   1:  PR[GP1:91,2] = PR[GP1:90,2] + 15.763;
   1:L PR[91] R[100]mm/sec CNT100;
   1:  PR[GP1:91,1] = PR[GP1:90,1] + -26.616;
   1:  PR[GP1:91,2] = PR[GP1:90,2] + 13.647;
   1:L PR[91] R[100]mm/sec CNT100;
   1:  PR[GP1:91,1] = PR[GP1:90,1] + -28.624;
   1:  PR[GP1:91,2] = PR[GP1:90,2] + 11.003;
   1:L PR[91] R[100]mm/sec CNT100;
   1:  PR[GP1:91,1] = PR[GP1:90,1] + -29.736;
   1:  PR[GP1:91,2] = PR[GP1:90,2] + 8.431;
   1:L PR[91] R[100]mm/sec CNT100;
   1:  PR[GP1:91,1] = PR[GP1:90,1] + -30.927;
   1:  PR[GP1:91,2] = PR[GP1:90,2] + 5.553;
   1:L PR[91] R[100]mm/sec CNT100;
   1:  PR[GP1:91,1] = PR[GP1:90,1] + -31.315;
   1:  PR[GP1:91,2] = PR[GP1:90,2] + 2.689;
   1:L PR[91] R[100]mm/sec CNT100;
   1:  PR[GP1:91,1] = PR[GP1:90,1] + -31.610;
   1:  PR[GP1:91,2] = PR[GP1:90,2] + -0.285;
   1:L PR[91] R[100]mm/sec CNT100;
   1:  PR[GP1:91,1] = PR[GP1:90,1] + -31.568;
   1:  PR[GP1:91,2] = PR[GP1:90,2] + -0.593;
   1:L PR[91] R[100]mm/sec CNT100;
   1:  PR[GP1:91,1] = PR[GP1:90,1] + -31.320;
   1:  PR[GP1:91,2] = PR[GP1:90,2] + -3.189;
   1:L PR[91] R[100]mm/sec CNT100;
   1:  PR[GP1:91,1] = PR[GP1:90,1] + -30.924;
   1:  PR[GP1:91,2] = PR[GP1:90,2] + -6.186;
   1:L PR[91] R[100]mm/sec CNT100;
   1:  PR[GP1:91,1] = PR[GP1:90,1] + -29.732;
   1:  PR[GP1:91,2] = PR[GP1:90,2] + -9.064;
   1:L PR[91] R[100]mm/sec CNT100;
   1:  PR[GP1:91,1] = PR[GP1:90,1] + -28.617;
   1:  PR[GP1:91,2] = PR[GP1:90,2] + -11.639;
   1:L PR[91] R[100]mm/sec CNT100;
   1:  PR[GP1:91,1] = PR[GP1:90,1] + -26.605;
   1:  PR[GP1:91,2] = PR[GP1:90,2] + -14.284;
   1:L PR[91] R[100]mm/sec CNT100;
   1:  PR[GP1:91,1] = PR[GP1:90,1] + -24.927;
   1:  PR[GP1:91,2] = PR[GP1:90,2] + -16.401;
   1:L PR[91] R[100]mm/sec CNT100;
   1:  PR[GP1:91,1] = PR[GP1:90,1] + -22.102;
   1:  PR[GP1:91,2] = PR[GP1:90,2] + -18.610;
   1:L PR[91] R[100]mm/sec CNT100;
   1:  PR[GP1:91,1] = PR[GP1:90,1] + -20.094;
   1:  PR[GP1:91,2] = PR[GP1:90,2] + -20.099;
   1:L PR[91] R[100]mm/sec CNT100;
   1:  PR[GP1:91,1] = PR[GP1:90,1] + -16.514;
   1:  PR[GP1:91,2] = PR[GP1:90,2] + -21.656;
   1:L PR[91] R[100]mm/sec CNT100;
   1:  PR[GP1:91,1] = PR[GP1:90,1] + -14.429;
   1:  PR[GP1:91,2] = PR[GP1:90,2] + -22.497;
   1:L PR[91] R[100]mm/sec CNT100;
   1:  PR[GP1:91,1] = PR[GP1:90,1] + -10.253;
   1:  PR[GP1:91,2] = PR[GP1:90,2] + -23.160;
   1:L PR[91] R[100]mm/sec CNT100;
   1:  PR[GP1:91,1] = PR[GP1:90,1] + -8.313;
   1:  PR[GP1:91,2] = PR[GP1:90,2] + -23.412;
   1:L PR[91] R[100]mm/sec CNT100;
   1:  PR[GP1:91,1] = PR[GP1:90,1] + -3.668;
   1:  PR[GP1:91,2] = PR[GP1:90,2] + -22.952;
   1:L PR[91] R[100]mm/sec CNT100;
   1:  PR[GP1:91,1] = PR[GP1:90,1] + -2.097;
   1:  PR[GP1:91,2] = PR[GP1:90,2] + -22.752;
   1:L PR[91] R[100]mm/sec CNT100;
   1:  PR[GP1:91,1] = PR[GP1:90,1] + -1.786;
   1:  PR[GP1:91,2] = PR[GP1:90,2] + -22.654;
   1:L PR[91] R[100]mm/sec CNT100;
   1:  PR[GP1:91,1] = PR[GP1:90,1] + -0.630;
   1:  PR[GP1:91,2] = PR[GP1:90,2] + -22.246;
   1:L PR[91] R[100]mm/sec CNT100;
   1:  PR[GP1:91,1] = PR[GP1:90,1] + 0.801;
   1:  PR[GP1:91,2] = PR[GP1:90,2] + -22.273;
   1:L PR[91] R[100]mm/sec CNT100;
   1:  PR[GP1:91,1] = PR[GP1:90,1] + 1.811;
   1:  PR[GP1:91,2] = PR[GP1:90,2] + -22.609;
   1:L PR[91] R[100]mm/sec CNT100;
   1:  PR[GP1:91,1] = PR[GP1:90,1] + 2.902;
   1:  PR[GP1:91,2] = PR[GP1:90,2] + -22.750;
   1:L PR[91] R[100]mm/sec CNT100;
   1:  PR[GP1:91,1] = PR[GP1:90,1] + 3.884;
   1:  PR[GP1:91,2] = PR[GP1:90,2] + -22.958;
   1:L PR[91] R[100]mm/sec CNT100;
   1:  PR[GP1:91,1] = PR[GP1:90,1] + 8.470;
   1:  PR[GP1:91,2] = PR[GP1:90,2] + -23.412;
   1:L PR[91] R[100]mm/sec CNT100;
   1:  PR[GP1:91,1] = PR[GP1:90,1] + 10.410;
   1:  PR[GP1:91,2] = PR[GP1:90,2] + -23.160;
   1:L PR[91] R[100]mm/sec CNT100;
   1:  PR[GP1:91,1] = PR[GP1:90,1] + 14.586;
   1:  PR[GP1:91,2] = PR[GP1:90,2] + -22.496;
   1:L PR[91] R[100]mm/sec CNT100;
   1:  PR[GP1:91,1] = PR[GP1:90,1] + 16.671;
   1:  PR[GP1:91,2] = PR[GP1:90,2] + -21.656;
   1:L PR[91] R[100]mm/sec CNT100;
   1:  PR[GP1:91,1] = PR[GP1:90,1] + 20.251;
   1:  PR[GP1:91,2] = PR[GP1:90,2] + -20.100;
   1:L PR[91] R[100]mm/sec CNT100;
   1:  PR[GP1:91,1] = PR[GP1:90,1] + 22.259;
   1:  PR[GP1:91,2] = PR[GP1:90,2] + -18.611;
   1:L PR[91] R[100]mm/sec CNT100;
   1:  PR[GP1:91,1] = PR[GP1:90,1] + 25.083;
   1:  PR[GP1:91,2] = PR[GP1:90,2] + -16.402;
   1:L PR[91] R[100]mm/sec CNT100;
   1:  PR[GP1:91,1] = PR[GP1:90,1] + 26.761;
   1:  PR[GP1:91,2] = PR[GP1:90,2] + -14.281;
   1:L PR[91] R[100]mm/sec CNT100;
   1:  PR[GP1:91,1] = PR[GP1:90,1] + 28.774;
   1:  PR[GP1:91,2] = PR[GP1:90,2] + -11.633;
   1:L PR[91] R[100]mm/sec CNT100;
   1:  PR[GP1:91,1] = PR[GP1:90,1] + 29.890;
   1:  PR[GP1:91,2] = PR[GP1:90,2] + -9.068;
   1:L PR[91] R[100]mm/sec CNT100;
   1:  PR[GP1:91,1] = PR[GP1:90,1] + 31.082;
   1:  PR[GP1:91,2] = PR[GP1:90,2] + -6.194;
   1:L PR[91] R[100]mm/sec CNT100;
   1:  PR[GP1:91,1] = PR[GP1:90,1] + 31.471;
   1:  PR[GP1:91,2] = PR[GP1:90,2] + -3.318;
   1:L PR[91] R[100]mm/sec CNT100;
   1:  PR[GP1:91,1] = PR[GP1:90,1] + 31.767;
   1:  PR[GP1:91,2] = PR[GP1:90,2] + -0.338;
   1:L PR[91] R[100]mm/sec CNT100;
   1:  PR[GP1:91,1] = PR[GP1:90,1] + 31.725;
   1:  PR[GP1:91,2] = PR[GP1:90,2] + -0.030;
   1:L PR[91] R[100]mm/sec CNT100;
   1:  PR[GP1:91,1] = PR[GP1:90,1] + 31.477;
   1:  PR[GP1:91,2] = PR[GP1:90,2] + 2.571;
   1:L PR[91] R[100]mm/sec CNT100;
   1:  PR[GP1:91,1] = PR[GP1:90,1] + 31.083;
   1:  PR[GP1:91,2] = PR[GP1:90,2] + 5.567;
   1:L PR[91] R[100]mm/sec CNT100;
   1:  PR[GP1:91,1] = PR[GP1:90,1] + 29.894;
   1:  PR[GP1:91,2] = PR[GP1:90,2] + 8.436;
   1:L PR[91] R[100]mm/sec CNT100;
   1:  PR[GP1:91,1] = PR[GP1:90,1] + 28.781;
   1:  PR[GP1:91,2] = PR[GP1:90,2] + 10.998;
   1:L PR[91] R[100]mm/sec CNT100;
   1:  PR[GP1:91,1] = PR[GP1:90,1] + 26.772;
   1:  PR[GP1:91,2] = PR[GP1:90,2] + 13.644;
   1:L PR[91] R[100]mm/sec CNT100;
   1:  PR[GP1:91,1] = PR[GP1:90,1] + 25.097;
   1:  PR[GP1:91,2] = PR[GP1:90,2] + 15.764;
   1:L PR[91] R[100]mm/sec CNT100;
   1:  PR[GP1:91,1] = PR[GP1:90,1] + 22.278;
   1:  PR[GP1:91,2] = PR[GP1:90,2] + 17.973;
   1:L PR[91] R[100]mm/sec CNT100;
   1:  PR[GP1:91,1] = PR[GP1:90,1] + 20.273;
   1:  PR[GP1:91,2] = PR[GP1:90,2] + 19.463;
   1:L PR[91] R[100]mm/sec CNT100;
   1:  PR[GP1:91,1] = PR[GP1:90,1] + 16.700;
   1:  PR[GP1:91,2] = PR[GP1:90,2] + 21.021;
   1:L PR[91] R[100]mm/sec CNT100;
   1:  PR[GP1:91,1] = PR[GP1:90,1] + 14.617;
   1:  PR[GP1:91,2] = PR[GP1:90,2] + 21.864;
   1:L PR[91] R[100]mm/sec CNT100;
   1:  PR[GP1:91,1] = PR[GP1:90,1] + 10.447;
   1:  PR[GP1:91,2] = PR[GP1:90,2] + 22.532;
   1:L PR[91] R[100]mm/sec CNT100;
   1:  PR[GP1:91,1] = PR[GP1:90,1] + 8.508;
   1:  PR[GP1:91,2] = PR[GP1:90,2] + 22.787;
   1:L PR[91] R[100]mm/sec CNT100;
   1:  PR[GP1:91,1] = PR[GP1:90,1] + 3.910;
   1:  PR[GP1:91,2] = PR[GP1:90,2] + 22.344;
   1:L PR[91] R[100]mm/sec CNT100;
   1:  PR[GP1:91,1] = PR[GP1:90,1] + 2.308;
   1:  PR[GP1:91,2] = PR[GP1:90,2] + 22.142;
   1:L PR[91] R[100]mm/sec CNT100;
   1:  PR[GP1:91,1] = PR[GP1:90,1] + 0.792;
   1:  PR[GP1:91,2] = PR[GP1:90,2] + 21.648;
   1:L PR[91] R[100]mm/sec CNT100;
   1:  PR[91] = PR[90];
   1:  PR[GP1:91,1] = PR[GP1:90,1] + -0.605;
   1:  PR[GP1:91,2] = PR[GP1:90,2] + 21.812;
   1:  PR[GP1:91,3] = PR[GP1:90,3] + 53.985;
   1:L PR[91] R[100]mm/sec CNT100;
   1:  PR[GP1:91,1] = PR[GP1:90,1] + -1.935;
   1:  PR[GP1:91,2] = PR[GP1:90,2] + 22.247;
   1:L PR[91] R[100]mm/sec CNT100;
   1:  PR[GP1:91,1] = PR[GP1:90,1] + -3.290;
   1:  PR[GP1:91,2] = PR[GP1:90,2] + 22.418;
   1:L PR[91] R[100]mm/sec CNT100;
   1:  PR[GP1:91,1] = PR[GP1:90,1] + -8.152;
   1:  PR[GP1:91,2] = PR[GP1:90,2] + 22.887;
   1:L PR[91] R[100]mm/sec CNT100;
   1:  PR[GP1:91,1] = PR[GP1:90,1] + -9.841;
   1:  PR[GP1:91,2] = PR[GP1:90,2] + 22.665;
   1:L PR[91] R[100]mm/sec CNT100;
   1:  PR[GP1:91,1] = PR[GP1:90,1] + -14.276;
   1:  PR[GP1:91,2] = PR[GP1:90,2] + 21.954;
   1:L PR[91] R[100]mm/sec CNT100;
   1:  PR[GP1:91,1] = PR[GP1:90,1] + -16.118;
   1:  PR[GP1:91,2] = PR[GP1:90,2] + 21.208;
   1:L PR[91] R[100]mm/sec CNT100;
   1:  PR[GP1:91,1] = PR[GP1:90,1] + -19.944;
   1:  PR[GP1:91,2] = PR[GP1:90,2] + 19.539;
   1:L PR[91] R[100]mm/sec CNT100;
   1:  PR[GP1:91,1] = PR[GP1:90,1] + -21.739;
   1:  PR[GP1:91,2] = PR[GP1:90,2] + 18.205;
   1:L PR[91] R[100]mm/sec CNT100;
   1:  PR[GP1:91,1] = PR[GP1:90,1] + -24.778;
   1:  PR[GP1:91,2] = PR[GP1:90,2] + 15.824;
   1:L PR[91] R[100]mm/sec CNT100;
   1:  PR[GP1:91,1] = PR[GP1:90,1] + -26.290;
   1:  PR[GP1:91,2] = PR[GP1:90,2] + 13.915;
   1:L PR[91] R[100]mm/sec CNT100;
   1:  PR[GP1:91,1] = PR[GP1:90,1] + -28.469;
   1:  PR[GP1:91,2] = PR[GP1:90,2] + 11.046;
   1:L PR[91] R[100]mm/sec CNT100;
   1:  PR[GP1:91,1] = PR[GP1:90,1] + -29.478;
   1:  PR[GP1:91,2] = PR[GP1:90,2] + 8.712;
   1:L PR[91] R[100]mm/sec CNT100;
   1:  PR[GP1:91,1] = PR[GP1:90,1] + -30.777;
   1:  PR[GP1:91,2] = PR[GP1:90,2] + 5.574;
   1:L PR[91] R[100]mm/sec CNT100;
   1:  PR[GP1:91,1] = PR[GP1:90,1] + -31.130;
   1:  PR[GP1:91,2] = PR[GP1:90,2] + 2.970;
   1:L PR[91] R[100]mm/sec CNT100;
   1:  PR[GP1:91,1] = PR[GP1:90,1] + -31.456;
   1:  PR[GP1:91,2] = PR[GP1:90,2] + -0.315;
   1:L PR[91] R[100]mm/sec CNT100;
   1:  PR[GP1:91,1] = PR[GP1:90,1] + -31.205;
   1:  PR[GP1:91,2] = PR[GP1:90,2] + -2.938;
   1:L PR[91] R[100]mm/sec CNT100;
   1:  PR[GP1:91,1] = PR[GP1:90,1] + -30.774;
   1:  PR[GP1:91,2] = PR[GP1:90,2] + -6.207;
   1:L PR[91] R[100]mm/sec CNT100;
   1:  PR[GP1:91,1] = PR[GP1:90,1] + -29.474;
   1:  PR[GP1:91,2] = PR[GP1:90,2] + -9.345;
   1:L PR[91] R[100]mm/sec CNT100;
   1:  PR[GP1:91,1] = PR[GP1:90,1] + -28.462;
   1:  PR[GP1:91,2] = PR[GP1:90,2] + -11.681;
   1:L PR[91] R[100]mm/sec CNT100;
   1:  PR[GP1:91,1] = PR[GP1:90,1] + -26.279;
   1:  PR[GP1:91,2] = PR[GP1:90,2] + -14.552;
   1:L PR[91] R[100]mm/sec CNT100;
   1:  PR[GP1:91,1] = PR[GP1:90,1] + -24.765;
   1:  PR[GP1:91,2] = PR[GP1:90,2] + -16.462;
   1:L PR[91] R[100]mm/sec CNT100;
   1:  PR[GP1:91,1] = PR[GP1:90,1] + -21.719;
   1:  PR[GP1:91,2] = PR[GP1:90,2] + -18.843;
   1:L PR[91] R[100]mm/sec CNT100;
   1:  PR[GP1:91,1] = PR[GP1:90,1] + -19.922;
   1:  PR[GP1:91,2] = PR[GP1:90,2] + -20.176;
   1:L PR[91] R[100]mm/sec CNT100;
   1:  PR[GP1:91,1] = PR[GP1:90,1] + -16.089;
   1:  PR[GP1:91,2] = PR[GP1:90,2] + -21.843;
   1:L PR[91] R[100]mm/sec CNT100;
   1:  PR[GP1:91,1] = PR[GP1:90,1] + -14.245;
   1:  PR[GP1:91,2] = PR[GP1:90,2] + -22.587;
   1:L PR[91] R[100]mm/sec CNT100;
   1:  PR[GP1:91,1] = PR[GP1:90,1] + -9.803;
   1:  PR[GP1:91,2] = PR[GP1:90,2] + -23.292;
   1:L PR[91] R[100]mm/sec CNT100;
   1:  PR[GP1:91,1] = PR[GP1:90,1] + -8.114;
   1:  PR[GP1:91,2] = PR[GP1:90,2] + -23.511;
   1:L PR[91] R[100]mm/sec CNT100;
   1:  PR[GP1:91,1] = PR[GP1:90,1] + -3.203;
   1:  PR[GP1:91,2] = PR[GP1:90,2] + -23.026;
   1:L PR[91] R[100]mm/sec CNT100;
   1:  PR[GP1:91,1] = PR[GP1:90,1] + -1.881;
   1:  PR[GP1:91,2] = PR[GP1:90,2] + -22.857;
   1:L PR[91] R[100]mm/sec CNT100;
   1:  PR[GP1:91,1] = PR[GP1:90,1] + -1.546;
   1:  PR[GP1:91,2] = PR[GP1:90,2] + -22.752;
   1:L PR[91] R[100]mm/sec CNT100;
   1:  PR[GP1:91,1] = PR[GP1:90,1] + -0.617;
   1:  PR[GP1:91,2] = PR[GP1:90,2] + -22.424;
   1:L PR[91] R[100]mm/sec CNT100;
   1:  PR[GP1:91,1] = PR[GP1:90,1] + 0.783;
   1:  PR[GP1:91,2] = PR[GP1:90,2] + -22.445;
   1:L PR[91] R[100]mm/sec CNT100;
   1:  PR[GP1:91,1] = PR[GP1:90,1] + 1.572;
   1:  PR[GP1:91,2] = PR[GP1:90,2] + -22.707;
   1:L PR[91] R[100]mm/sec CNT100;
   1:  PR[GP1:91,1] = PR[GP1:90,1] + 2.382;
   1:  PR[GP1:91,2] = PR[GP1:90,2] + -22.812;
   1:L PR[91] R[100]mm/sec CNT100;
   1:  PR[GP1:91,1] = PR[GP1:90,1] + 3.419;
   1:  PR[GP1:91,2] = PR[GP1:90,2] + -23.032;
   1:L PR[91] R[100]mm/sec CNT100;
   1:  PR[GP1:91,1] = PR[GP1:90,1] + 8.272;
   1:  PR[GP1:91,2] = PR[GP1:90,2] + -23.511;
   1:L PR[91] R[100]mm/sec CNT100;
   1:  PR[GP1:91,1] = PR[GP1:90,1] + 9.961;
   1:  PR[GP1:91,2] = PR[GP1:90,2] + -23.292;
   1:L PR[91] R[100]mm/sec CNT100;
   1:  PR[GP1:91,1] = PR[GP1:90,1] + 14.402;
   1:  PR[GP1:91,2] = PR[GP1:90,2] + -22.586;
   1:L PR[91] R[100]mm/sec CNT100;
   1:  PR[GP1:91,1] = PR[GP1:90,1] + 16.247;
   1:  PR[GP1:91,2] = PR[GP1:90,2] + -21.843;
   1:L PR[91] R[100]mm/sec CNT100;
   1:  PR[GP1:91,1] = PR[GP1:90,1] + 20.079;
   1:  PR[GP1:91,2] = PR[GP1:90,2] + -20.176;
   1:L PR[91] R[100]mm/sec CNT100;
   1:  PR[GP1:91,1] = PR[GP1:90,1] + 21.876;
   1:  PR[GP1:91,2] = PR[GP1:90,2] + -18.844;
   1:L PR[91] R[100]mm/sec CNT100;
   1:  PR[GP1:91,1] = PR[GP1:90,1] + 24.921;
   1:  PR[GP1:91,2] = PR[GP1:90,2] + -16.462;
   1:L PR[91] R[100]mm/sec CNT100;
   1:  PR[GP1:91,1] = PR[GP1:90,1] + 26.436;
   1:  PR[GP1:91,2] = PR[GP1:90,2] + -14.549;
   1:L PR[91] R[100]mm/sec CNT100;
   1:  PR[GP1:91,1] = PR[GP1:90,1] + 28.620;
   1:  PR[GP1:91,2] = PR[GP1:90,2] + -11.676;
   1:L PR[91] R[100]mm/sec CNT100;
   1:  PR[GP1:91,1] = PR[GP1:90,1] + 29.631;
   1:  PR[GP1:91,2] = PR[GP1:90,2] + -9.349;
   1:L PR[91] R[100]mm/sec CNT100;
   1:  PR[GP1:91,1] = PR[GP1:90,1] + 30.932;
   1:  PR[GP1:91,2] = PR[GP1:90,2] + -6.215;
   1:L PR[91] R[100]mm/sec CNT100;
   1:  PR[GP1:91,1] = PR[GP1:90,1] + 31.286;
   1:  PR[GP1:91,2] = PR[GP1:90,2] + -3.600;
   1:L PR[91] R[100]mm/sec CNT100;
   1:  PR[GP1:91,1] = PR[GP1:90,1] + 31.613;
   1:  PR[GP1:91,2] = PR[GP1:90,2] + -0.309;
   1:L PR[91] R[100]mm/sec CNT100;
   1:  PR[GP1:91,1] = PR[GP1:90,1] + 31.363;
   1:  PR[GP1:91,2] = PR[GP1:90,2] + 2.319;
   1:L PR[91] R[100]mm/sec CNT100;
   1:  PR[GP1:91,1] = PR[GP1:90,1] + 30.932;
   1:  PR[GP1:91,2] = PR[GP1:90,2] + 5.587;
   1:L PR[91] R[100]mm/sec CNT100;
   1:  PR[GP1:91,1] = PR[GP1:90,1] + 29.635;
   1:  PR[GP1:91,2] = PR[GP1:90,2] + 8.716;
   1:L PR[91] R[100]mm/sec CNT100;
   1:  PR[GP1:91,1] = PR[GP1:90,1] + 28.626;
   1:  PR[GP1:91,2] = PR[GP1:90,2] + 11.041;
   1:L PR[91] R[100]mm/sec CNT100;
   1:  PR[GP1:91,1] = PR[GP1:90,1] + 26.446;
   1:  PR[GP1:91,2] = PR[GP1:90,2] + 13.912;
   1:L PR[91] R[100]mm/sec CNT100;
   1:  PR[GP1:91,1] = PR[GP1:90,1] + 24.934;
   1:  PR[GP1:91,2] = PR[GP1:90,2] + 15.825;
   1:L PR[91] R[100]mm/sec CNT100;
   1:  PR[GP1:91,1] = PR[GP1:90,1] + 21.896;
   1:  PR[GP1:91,2] = PR[GP1:90,2] + 18.206;
   1:L PR[91] R[100]mm/sec CNT100;
   1:  PR[GP1:91,1] = PR[GP1:90,1] + 20.101;
   1:  PR[GP1:91,2] = PR[GP1:90,2] + 19.540;
   1:L PR[91] R[100]mm/sec CNT100;
   1:  PR[GP1:91,1] = PR[GP1:90,1] + 16.275;
   1:  PR[GP1:91,2] = PR[GP1:90,2] + 21.208;
   1:L PR[91] R[100]mm/sec CNT100;
   1:  PR[GP1:91,1] = PR[GP1:90,1] + 14.433;
   1:  PR[GP1:91,2] = PR[GP1:90,2] + 21.953;
   1:L PR[91] R[100]mm/sec CNT100;
   1:  PR[GP1:91,1] = PR[GP1:90,1] + 9.998;
   1:  PR[GP1:91,2] = PR[GP1:90,2] + 22.665;
   1:L PR[91] R[100]mm/sec CNT100;
   1:  PR[GP1:91,1] = PR[GP1:90,1] + 8.309;
   1:  PR[GP1:91,2] = PR[GP1:90,2] + 22.887;
   1:L PR[91] R[100]mm/sec CNT100;
   1:  PR[GP1:91,1] = PR[GP1:90,1] + 3.448;
   1:  PR[GP1:91,2] = PR[GP1:90,2] + 22.418;
   1:L PR[91] R[100]mm/sec CNT100;
   1:  PR[GP1:91,1] = PR[GP1:90,1] + 2.090;
   1:  PR[GP1:91,2] = PR[GP1:90,2] + 22.247;
   1:L PR[91] R[100]mm/sec CNT100;
   1:  PR[GP1:91,1] = PR[GP1:90,1] + 0.770;
   1:  PR[GP1:91,2] = PR[GP1:90,2] + 21.820;
   1:L PR[91] R[100]mm/sec CNT100;
   1:  PR[91] = PR[90];
   1:  PR[GP1:91,1] = PR[GP1:90,1] + -0.589;
   1:  PR[GP1:91,2] = PR[GP1:90,2] + 21.992;
   1:  PR[GP1:91,3] = PR[GP1:90,3] + 54.595;
   1:L PR[91] R[100]mm/sec CNT100;
   1:  PR[GP1:91,1] = PR[GP1:90,1] + -1.714;
   1:  PR[GP1:91,2] = PR[GP1:90,2] + 22.352;
   1:L PR[91] R[100]mm/sec CNT100;
   1:  PR[GP1:91,1] = PR[GP1:90,1] + -2.827;
   1:  PR[GP1:91,2] = PR[GP1:90,2] + 22.492;
   1:L PR[91] R[100]mm/sec CNT100;
   1:  PR[GP1:91,1] = PR[GP1:90,1] + -7.953;
   1:  PR[GP1:91,2] = PR[GP1:90,2] + 22.986;
   1:L PR[91] R[100]mm/sec CNT100;
   1:  PR[GP1:91,1] = PR[GP1:90,1] + -9.391;
   1:  PR[GP1:91,2] = PR[GP1:90,2] + 22.797;
   1:L PR[91] R[100]mm/sec CNT100;
   1:  PR[GP1:91,1] = PR[GP1:90,1] + -14.091;
   1:  PR[GP1:91,2] = PR[GP1:90,2] + 22.044;
   1:L PR[91] R[100]mm/sec CNT100;
   1:  PR[GP1:91,1] = PR[GP1:90,1] + -15.693;
   1:  PR[GP1:91,2] = PR[GP1:90,2] + 21.395;
   1:L PR[91] R[100]mm/sec CNT100;
   1:  PR[GP1:91,1] = PR[GP1:90,1] + -19.772;
   1:  PR[GP1:91,2] = PR[GP1:90,2] + 19.616;
   1:L PR[91] R[100]mm/sec CNT100;
   1:  PR[GP1:91,1] = PR[GP1:90,1] + -21.356;
   1:  PR[GP1:91,2] = PR[GP1:90,2] + 18.438;
   1:L PR[91] R[100]mm/sec CNT100;
   1:  PR[GP1:91,1] = PR[GP1:90,1] + -24.616;
   1:  PR[GP1:91,2] = PR[GP1:90,2] + 15.885;
   1:L PR[91] R[100]mm/sec CNT100;
   1:  PR[GP1:91,1] = PR[GP1:90,1] + -25.964;
   1:  PR[GP1:91,2] = PR[GP1:90,2] + 14.182;
   1:L PR[91] R[100]mm/sec CNT100;
   1:  PR[GP1:91,1] = PR[GP1:90,1] + -28.314;
   1:  PR[GP1:91,2] = PR[GP1:90,2] + 11.088;
   1:L PR[91] R[100]mm/sec CNT100;
   1:  PR[GP1:91,1] = PR[GP1:90,1] + -29.220;
   1:  PR[GP1:91,2] = PR[GP1:90,2] + 8.993;
   1:L PR[91] R[100]mm/sec CNT100;
   1:  PR[GP1:91,1] = PR[GP1:90,1] + -30.626;
   1:  PR[GP1:91,2] = PR[GP1:90,2] + 5.595;
   1:L PR[91] R[100]mm/sec CNT100;
   1:  PR[GP1:91,1] = PR[GP1:90,1] + -30.944;
   1:  PR[GP1:91,2] = PR[GP1:90,2] + 3.251;
   1:L PR[91] R[100]mm/sec CNT100;
   1:  PR[GP1:91,1] = PR[GP1:90,1] + -31.251;
   1:  PR[GP1:91,2] = PR[GP1:90,2] + 0.151;
   1:L PR[91] R[100]mm/sec CNT100;
   1:  PR[GP1:91,1] = PR[GP1:90,1] + -31.315;
   1:  PR[GP1:91,2] = PR[GP1:90,2] + -0.338;
   1:L PR[91] R[100]mm/sec CNT100;
   1:  PR[GP1:91,1] = PR[GP1:90,1] + -31.091;
   1:  PR[GP1:91,2] = PR[GP1:90,2] + -2.686;
   1:L PR[91] R[100]mm/sec CNT100;
   1:  PR[GP1:91,1] = PR[GP1:90,1] + -30.623;
   1:  PR[GP1:91,2] = PR[GP1:90,2] + -6.228;
   1:L PR[91] R[100]mm/sec CNT100;
   1:  PR[GP1:91,1] = PR[GP1:90,1] + -29.215;
   1:  PR[GP1:91,2] = PR[GP1:90,2] + -9.626;
   1:L PR[91] R[100]mm/sec CNT100;
   1:  PR[GP1:91,1] = PR[GP1:90,1] + -28.307;
   1:  PR[GP1:91,2] = PR[GP1:90,2] + -11.724;
   1:L PR[91] R[100]mm/sec CNT100;
   1:  PR[GP1:91,1] = PR[GP1:90,1] + -25.953;
   1:  PR[GP1:91,2] = PR[GP1:90,2] + -14.819;
   1:L PR[91] R[100]mm/sec CNT100;
   1:  PR[GP1:91,1] = PR[GP1:90,1] + -24.602;
   1:  PR[GP1:91,2] = PR[GP1:90,2] + -16.522;
   1:L PR[91] R[100]mm/sec CNT100;
   1:  PR[GP1:91,1] = PR[GP1:90,1] + -21.336;
   1:  PR[GP1:91,2] = PR[GP1:90,2] + -19.076;
   1:L PR[91] R[100]mm/sec CNT100;
   1:  PR[GP1:91,1] = PR[GP1:90,1] + -19.750;
   1:  PR[GP1:91,2] = PR[GP1:90,2] + -20.253;
   1:L PR[91] R[100]mm/sec CNT100;
   1:  PR[GP1:91,1] = PR[GP1:90,1] + -15.664;
   1:  PR[GP1:91,2] = PR[GP1:90,2] + -22.030;
   1:L PR[91] R[100]mm/sec CNT100;
   1:  PR[GP1:91,1] = PR[GP1:90,1] + -14.061;
   1:  PR[GP1:91,2] = PR[GP1:90,2] + -22.677;
   1:L PR[91] R[100]mm/sec CNT100;
   1:  PR[GP1:91,1] = PR[GP1:90,1] + -9.354;
   1:  PR[GP1:91,2] = PR[GP1:90,2] + -23.424;
   1:L PR[91] R[100]mm/sec CNT100;
   1:  PR[GP1:91,1] = PR[GP1:90,1] + -7.915;
   1:  PR[GP1:91,2] = PR[GP1:90,2] + -23.611;
   1:L PR[91] R[100]mm/sec CNT100;
   1:  PR[GP1:91,1] = PR[GP1:90,1] + -2.738;
   1:  PR[GP1:91,2] = PR[GP1:90,2] + -23.099;
   1:L PR[91] R[100]mm/sec CNT100;
   1:  PR[GP1:91,1] = PR[GP1:90,1] + -1.676;
   1:  PR[GP1:91,2] = PR[GP1:90,2] + -22.963;
   1:L PR[91] R[100]mm/sec CNT100;
   1:  PR[GP1:91,1] = PR[GP1:90,1] + -0.592;
   1:  PR[GP1:91,2] = PR[GP1:90,2] + -22.602;
   1:L PR[91] R[100]mm/sec CNT100;
   1:  PR[GP1:91,1] = PR[GP1:90,1] + 0.765;
   1:  PR[GP1:91,2] = PR[GP1:90,2] + -22.616;
   1:L PR[91] R[100]mm/sec CNT100;
   1:  PR[GP1:91,1] = PR[GP1:90,1] + 1.333;
   1:  PR[GP1:91,2] = PR[GP1:90,2] + -22.805;
   1:L PR[91] R[100]mm/sec CNT100;
   1:  PR[GP1:91,1] = PR[GP1:90,1] + 1.862;
   1:  PR[GP1:91,2] = PR[GP1:90,2] + -22.874;
   1:L PR[91] R[100]mm/sec CNT100;
   1:  PR[GP1:91,1] = PR[GP1:90,1] + 2.955;
   1:  PR[GP1:91,2] = PR[GP1:90,2] + -23.105;
   1:L PR[91] R[100]mm/sec CNT100;
   1:  PR[GP1:91,1] = PR[GP1:90,1] + 8.073;
   1:  PR[GP1:91,2] = PR[GP1:90,2] + -23.611;
   1:L PR[91] R[100]mm/sec CNT100;
   1:  PR[GP1:91,1] = PR[GP1:90,1] + 9.512;
   1:  PR[GP1:91,2] = PR[GP1:90,2] + -23.424;
   1:L PR[91] R[100]mm/sec CNT100;
   1:  PR[GP1:91,1] = PR[GP1:90,1] + 14.218;
   1:  PR[GP1:91,2] = PR[GP1:90,2] + -22.676;
   1:L PR[91] R[100]mm/sec CNT100;
   1:  PR[GP1:91,1] = PR[GP1:90,1] + 15.823;
   1:  PR[GP1:91,2] = PR[GP1:90,2] + -22.030;
   1:L PR[91] R[100]mm/sec CNT100;
   1:  PR[GP1:91,1] = PR[GP1:90,1] + 19.907;
   1:  PR[GP1:91,2] = PR[GP1:90,2] + -20.253;
   1:L PR[91] R[100]mm/sec CNT100;
   1:  PR[GP1:91,1] = PR[GP1:90,1] + 21.493;
   1:  PR[GP1:91,2] = PR[GP1:90,2] + -19.077;
   1:L PR[91] R[100]mm/sec CNT100;
   1:  PR[GP1:91,1] = PR[GP1:90,1] + 24.759;
   1:  PR[GP1:91,2] = PR[GP1:90,2] + -16.523;
   1:L PR[91] R[100]mm/sec CNT100;
   1:  PR[GP1:91,1] = PR[GP1:90,1] + 26.110;
   1:  PR[GP1:91,2] = PR[GP1:90,2] + -14.816;
   1:L PR[91] R[100]mm/sec CNT100;
   1:  PR[GP1:91,1] = PR[GP1:90,1] + 28.465;
   1:  PR[GP1:91,2] = PR[GP1:90,2] + -11.718;
   1:L PR[91] R[100]mm/sec CNT100;
   1:  PR[GP1:91,1] = PR[GP1:90,1] + 29.373;
   1:  PR[GP1:91,2] = PR[GP1:90,2] + -9.630;
   1:L PR[91] R[100]mm/sec CNT100;
   1:  PR[GP1:91,1] = PR[GP1:90,1] + 30.781;
   1:  PR[GP1:91,2] = PR[GP1:90,2] + -6.235;
   1:L PR[91] R[100]mm/sec CNT100;
   1:  PR[GP1:91,1] = PR[GP1:90,1] + 31.100;
   1:  PR[GP1:91,2] = PR[GP1:90,2] + -3.881;
   1:L PR[91] R[100]mm/sec CNT100;
   1:  PR[GP1:91,1] = PR[GP1:90,1] + 31.408;
   1:  PR[GP1:91,2] = PR[GP1:90,2] + -0.776;
   1:L PR[91] R[100]mm/sec CNT100;
   1:  PR[GP1:91,1] = PR[GP1:90,1] + 31.472;
   1:  PR[GP1:91,2] = PR[GP1:90,2] + -0.286;
   1:L PR[91] R[100]mm/sec CNT100;
   1:  PR[GP1:91,1] = PR[GP1:90,1] + 31.248;
   1:  PR[GP1:91,2] = PR[GP1:90,2] + 2.066;
   1:L PR[91] R[100]mm/sec CNT100;
   1:  PR[GP1:91,1] = PR[GP1:90,1] + 30.782;
   1:  PR[GP1:91,2] = PR[GP1:90,2] + 5.608;
   1:L PR[91] R[100]mm/sec CNT100;
   1:  PR[GP1:91,1] = PR[GP1:90,1] + 29.377;
   1:  PR[GP1:91,2] = PR[GP1:90,2] + 8.997;
   1:L PR[91] R[100]mm/sec CNT100;
   1:  PR[GP1:91,1] = PR[GP1:90,1] + 28.471;
   1:  PR[GP1:91,2] = PR[GP1:90,2] + 11.083;
   1:L PR[91] R[100]mm/sec CNT100;
   1:  PR[GP1:91,1] = PR[GP1:90,1] + 26.120;
   1:  PR[GP1:91,2] = PR[GP1:90,2] + 14.180;
   1:L PR[91] R[100]mm/sec CNT100;
   1:  PR[GP1:91,1] = PR[GP1:90,1] + 24.772;
   1:  PR[GP1:91,2] = PR[GP1:90,2] + 15.886;
   1:L PR[91] R[100]mm/sec CNT100;
   1:  PR[GP1:91,1] = PR[GP1:90,1] + 21.513;
   1:  PR[GP1:91,2] = PR[GP1:90,2] + 18.439;
   1:L PR[91] R[100]mm/sec CNT100;
   1:  PR[GP1:91,1] = PR[GP1:90,1] + 19.929;
   1:  PR[GP1:91,2] = PR[GP1:90,2] + 19.617;
   1:L PR[91] R[100]mm/sec CNT100;
   1:  PR[GP1:91,1] = PR[GP1:90,1] + 15.851;
   1:  PR[GP1:91,2] = PR[GP1:90,2] + 21.395;
   1:L PR[91] R[100]mm/sec CNT100;
   1:  PR[GP1:91,1] = PR[GP1:90,1] + 14.248;
   1:  PR[GP1:91,2] = PR[GP1:90,2] + 22.043;
   1:L PR[91] R[100]mm/sec CNT100;
   1:  PR[GP1:91,1] = PR[GP1:90,1] + 9.549;
   1:  PR[GP1:91,2] = PR[GP1:90,2] + 22.797;
   1:L PR[91] R[100]mm/sec CNT100;
   1:  PR[GP1:91,1] = PR[GP1:90,1] + 8.110;
   1:  PR[GP1:91,2] = PR[GP1:90,2] + 22.986;
   1:L PR[91] R[100]mm/sec CNT100;
   1:  PR[GP1:91,1] = PR[GP1:90,1] + 2.985;
   1:  PR[GP1:91,2] = PR[GP1:90,2] + 22.492;
   1:L PR[91] R[100]mm/sec CNT100;
   1:  PR[GP1:91,1] = PR[GP1:90,1] + 1.872;
   1:  PR[GP1:91,2] = PR[GP1:90,2] + 22.351;
   1:L PR[91] R[100]mm/sec CNT100;
   1:  PR[GP1:91,1] = PR[GP1:90,1] + 0.749;
   1:  PR[GP1:91,2] = PR[GP1:90,2] + 21.992;
   1:L PR[91] R[100]mm/sec CNT100;
   1:  PR[91] = PR[90];
   1:  PR[GP1:91,1] = PR[GP1:90,1] + -0.574;
   1:  PR[GP1:91,2] = PR[GP1:90,2] + 22.162;
   1:  PR[GP1:91,3] = PR[GP1:90,3] + 55.205;
   1:L PR[91] R[100]mm/sec CNT100;
   1:  PR[GP1:91,1] = PR[GP1:90,1] + -1.497;
   1:  PR[GP1:91,2] = PR[GP1:90,2] + 22.457;
   1:L PR[91] R[100]mm/sec CNT100;
   1:  PR[GP1:91,1] = PR[GP1:90,1] + -2.364;
   1:  PR[GP1:91,2] = PR[GP1:90,2] + 22.566;
   1:L PR[91] R[100]mm/sec CNT100;
   1:  PR[GP1:91,1] = PR[GP1:90,1] + -7.753;
   1:  PR[GP1:91,2] = PR[GP1:90,2] + 23.086;
   1:L PR[91] R[100]mm/sec CNT100;
   1:  PR[GP1:91,1] = PR[GP1:90,1] + -8.942;
   1:  PR[GP1:91,2] = PR[GP1:90,2] + 22.929;
   1:L PR[91] R[100]mm/sec CNT100;
   1:  PR[GP1:91,1] = PR[GP1:90,1] + -13.907;
   1:  PR[GP1:91,2] = PR[GP1:90,2] + 22.134;
   1:L PR[91] R[100]mm/sec CNT100;
   1:  PR[GP1:91,1] = PR[GP1:90,1] + -15.269;
   1:  PR[GP1:91,2] = PR[GP1:90,2] + 21.582;
   1:L PR[91] R[100]mm/sec CNT100;
   1:  PR[GP1:91,1] = PR[GP1:90,1] + -19.600;
   1:  PR[GP1:91,2] = PR[GP1:90,2] + 19.693;
   1:L PR[91] R[100]mm/sec CNT100;
   1:  PR[GP1:91,1] = PR[GP1:90,1] + -20.974;
   1:  PR[GP1:91,2] = PR[GP1:90,2] + 18.672;
   1:L PR[91] R[100]mm/sec CNT100;
   1:  PR[GP1:91,1] = PR[GP1:90,1] + -24.454;
   1:  PR[GP1:91,2] = PR[GP1:90,2] + 15.946;
   1:L PR[91] R[100]mm/sec CNT100;
   1:  PR[GP1:91,1] = PR[GP1:90,1] + -25.638;
   1:  PR[GP1:91,2] = PR[GP1:90,2] + 14.449;
   1:L PR[91] R[100]mm/sec CNT100;
   1:  PR[GP1:91,1] = PR[GP1:90,1] + -28.159;
   1:  PR[GP1:91,2] = PR[GP1:90,2] + 11.131;
   1:L PR[91] R[100]mm/sec CNT100;
   1:  PR[GP1:91,1] = PR[GP1:90,1] + -28.962;
   1:  PR[GP1:91,2] = PR[GP1:90,2] + 9.274;
   1:L PR[91] R[100]mm/sec CNT100;
   1:  PR[GP1:91,1] = PR[GP1:90,1] + -30.476;
   1:  PR[GP1:91,2] = PR[GP1:90,2] + 5.616;
   1:L PR[91] R[100]mm/sec CNT100;
   1:  PR[GP1:91,1] = PR[GP1:90,1] + -30.758;
   1:  PR[GP1:91,2] = PR[GP1:90,2] + 3.532;
   1:L PR[91] R[100]mm/sec CNT100;
   1:  PR[GP1:91,1] = PR[GP1:90,1] + -31.034;
   1:  PR[GP1:91,2] = PR[GP1:90,2] + 0.748;
   1:L PR[91] R[100]mm/sec CNT100;
   1:  PR[GP1:91,1] = PR[GP1:90,1] + -31.177;
   1:  PR[GP1:91,2] = PR[GP1:90,2] + -0.338;
   1:L PR[91] R[100]mm/sec CNT100;
   1:  PR[GP1:91,1] = PR[GP1:90,1] + -30.976;
   1:  PR[GP1:91,2] = PR[GP1:90,2] + -2.434;
   1:L PR[91] R[100]mm/sec CNT100;
   1:  PR[GP1:91,1] = PR[GP1:90,1] + -30.473;
   1:  PR[GP1:91,2] = PR[GP1:90,2] + -6.249;
   1:L PR[91] R[100]mm/sec CNT100;
   1:  PR[GP1:91,1] = PR[GP1:90,1] + -28.957;
   1:  PR[GP1:91,2] = PR[GP1:90,2] + -9.907;
   1:L PR[91] R[100]mm/sec CNT100;
   1:  PR[GP1:91,1] = PR[GP1:90,1] + -28.152;
   1:  PR[GP1:91,2] = PR[GP1:90,2] + -11.766;
   1:L PR[91] R[100]mm/sec CNT100;
   1:  PR[GP1:91,1] = PR[GP1:90,1] + -25.627;
   1:  PR[GP1:91,2] = PR[GP1:90,2] + -15.086;
   1:L PR[91] R[100]mm/sec CNT100;
   1:  PR[GP1:91,1] = PR[GP1:90,1] + -24.440;
   1:  PR[GP1:91,2] = PR[GP1:90,2] + -16.583;
   1:L PR[91] R[100]mm/sec CNT100;
   1:  PR[GP1:91,1] = PR[GP1:90,1] + -20.954;
   1:  PR[GP1:91,2] = PR[GP1:90,2] + -19.309;
   1:L PR[91] R[100]mm/sec CNT100;
   1:  PR[GP1:91,1] = PR[GP1:90,1] + -19.578;
   1:  PR[GP1:91,2] = PR[GP1:90,2] + -20.330;
   1:L PR[91] R[100]mm/sec CNT100;
   1:  PR[GP1:91,1] = PR[GP1:90,1] + -15.240;
   1:  PR[GP1:91,2] = PR[GP1:90,2] + -22.217;
   1:L PR[91] R[100]mm/sec CNT100;
   1:  PR[GP1:91,1] = PR[GP1:90,1] + -13.876;
   1:  PR[GP1:91,2] = PR[GP1:90,2] + -22.767;
   1:L PR[91] R[100]mm/sec CNT100;
   1:  PR[GP1:91,1] = PR[GP1:90,1] + -8.905;
   1:  PR[GP1:91,2] = PR[GP1:90,2] + -23.557;
   1:L PR[91] R[100]mm/sec CNT100;
   1:  PR[GP1:91,1] = PR[GP1:90,1] + -7.716;
   1:  PR[GP1:91,2] = PR[GP1:90,2] + -23.710;
   1:L PR[91] R[100]mm/sec CNT100;
   1:  PR[GP1:91,1] = PR[GP1:90,1] + -2.273;
   1:  PR[GP1:91,2] = PR[GP1:90,2] + -23.172;
   1:L PR[91] R[100]mm/sec CNT100;
   1:  PR[GP1:91,1] = PR[GP1:90,1] + -1.456;
   1:  PR[GP1:91,2] = PR[GP1:90,2] + -23.068;
   1:L PR[91] R[100]mm/sec CNT100;
   1:  PR[GP1:91,1] = PR[GP1:90,1] + -0.575;
   1:  PR[GP1:91,2] = PR[GP1:90,2] + -22.780;
   1:L PR[91] R[100]mm/sec CNT100;
   1:  PR[GP1:91,1] = PR[GP1:90,1] + 0.746;
   1:  PR[GP1:91,2] = PR[GP1:90,2] + -22.787;
   1:L PR[91] R[100]mm/sec CNT100;
   1:  PR[GP1:91,1] = PR[GP1:90,1] + 1.094;
   1:  PR[GP1:91,2] = PR[GP1:90,2] + -22.903;
   1:L PR[91] R[100]mm/sec CNT100;
   1:  PR[GP1:91,1] = PR[GP1:90,1] + 1.342;
   1:  PR[GP1:91,2] = PR[GP1:90,2] + -22.935;
   1:L PR[91] R[100]mm/sec CNT100;
   1:  PR[GP1:91,1] = PR[GP1:90,1] + 2.490;
   1:  PR[GP1:91,2] = PR[GP1:90,2] + -23.178;
   1:L PR[91] R[100]mm/sec CNT100;
   1:  PR[GP1:91,1] = PR[GP1:90,1] + 7.874;
   1:  PR[GP1:91,2] = PR[GP1:90,2] + -23.711;
   1:L PR[91] R[100]mm/sec CNT100;
   1:  PR[GP1:91,1] = PR[GP1:90,1] + 9.063;
   1:  PR[GP1:91,2] = PR[GP1:90,2] + -23.557;
   1:L PR[91] R[100]mm/sec CNT100;
   1:  PR[GP1:91,1] = PR[GP1:90,1] + 14.034;
   1:  PR[GP1:91,2] = PR[GP1:90,2] + -22.766;
   1:L PR[91] R[100]mm/sec CNT100;
   1:  PR[GP1:91,1] = PR[GP1:90,1] + 15.398;
   1:  PR[GP1:91,2] = PR[GP1:90,2] + -22.216;
   1:L PR[91] R[100]mm/sec CNT100;
   1:  PR[GP1:91,1] = PR[GP1:90,1] + 19.735;
   1:  PR[GP1:91,2] = PR[GP1:90,2] + -20.330;
   1:L PR[91] R[100]mm/sec CNT100;
   1:  PR[GP1:91,1] = PR[GP1:90,1] + 21.111;
   1:  PR[GP1:91,2] = PR[GP1:90,2] + -19.310;
   1:L PR[91] R[100]mm/sec CNT100;
   1:  PR[GP1:91,1] = PR[GP1:90,1] + 24.597;
   1:  PR[GP1:91,2] = PR[GP1:90,2] + -16.584;
   1:L PR[91] R[100]mm/sec CNT100;
   1:  PR[GP1:91,1] = PR[GP1:90,1] + 25.784;
   1:  PR[GP1:91,2] = PR[GP1:90,2] + -15.084;
   1:L PR[91] R[100]mm/sec CNT100;
   1:  PR[GP1:91,1] = PR[GP1:90,1] + 28.310;
   1:  PR[GP1:91,2] = PR[GP1:90,2] + -11.761;
   1:L PR[91] R[100]mm/sec CNT100;
   1:  PR[GP1:91,1] = PR[GP1:90,1] + 29.115;
   1:  PR[GP1:91,2] = PR[GP1:90,2] + -9.910;
   1:L PR[91] R[100]mm/sec CNT100;
   1:  PR[GP1:91,1] = PR[GP1:90,1] + 30.631;
   1:  PR[GP1:91,2] = PR[GP1:90,2] + -6.256;
   1:L PR[91] R[100]mm/sec CNT100;
   1:  PR[GP1:91,1] = PR[GP1:90,1] + 30.914;
   1:  PR[GP1:91,2] = PR[GP1:90,2] + -4.163;
   1:L PR[91] R[100]mm/sec CNT100;
   1:  PR[GP1:91,1] = PR[GP1:90,1] + 31.190;
   1:  PR[GP1:91,2] = PR[GP1:90,2] + -1.374;
   1:L PR[91] R[100]mm/sec CNT100;
   1:  PR[GP1:91,1] = PR[GP1:90,1] + 31.333;
   1:  PR[GP1:91,2] = PR[GP1:90,2] + -0.286;
   1:L PR[91] R[100]mm/sec CNT100;
   1:  PR[GP1:91,1] = PR[GP1:90,1] + 31.133;
   1:  PR[GP1:91,2] = PR[GP1:90,2] + 1.814;
   1:L PR[91] R[100]mm/sec CNT100;
   1:  PR[GP1:91,1] = PR[GP1:90,1] + 30.631;
   1:  PR[GP1:91,2] = PR[GP1:90,2] + 5.628;
   1:L PR[91] R[100]mm/sec CNT100;
   1:  PR[GP1:91,1] = PR[GP1:90,1] + 29.119;
   1:  PR[GP1:91,2] = PR[GP1:90,2] + 9.277;
   1:L PR[91] R[100]mm/sec CNT100;
   1:  PR[GP1:91,1] = PR[GP1:90,1] + 28.316;
   1:  PR[GP1:91,2] = PR[GP1:90,2] + 11.126;
   1:L PR[91] R[100]mm/sec CNT100;
   1:  PR[GP1:91,1] = PR[GP1:90,1] + 25.795;
   1:  PR[GP1:91,2] = PR[GP1:90,2] + 14.447;
   1:L PR[91] R[100]mm/sec CNT100;
   1:  PR[GP1:91,1] = PR[GP1:90,1] + 24.610;
   1:  PR[GP1:91,2] = PR[GP1:90,2] + 15.946;
   1:L PR[91] R[100]mm/sec CNT100;
   1:  PR[GP1:91,1] = PR[GP1:90,1] + 21.131;
   1:  PR[GP1:91,2] = PR[GP1:90,2] + 18.672;
   1:L PR[91] R[100]mm/sec CNT100;
   1:  PR[GP1:91,1] = PR[GP1:90,1] + 19.757;
   1:  PR[GP1:91,2] = PR[GP1:90,2] + 19.693;
   1:L PR[91] R[100]mm/sec CNT100;
   1:  PR[GP1:91,1] = PR[GP1:90,1] + 15.427;
   1:  PR[GP1:91,2] = PR[GP1:90,2] + 21.582;
   1:L PR[91] R[100]mm/sec CNT100;
   1:  PR[GP1:91,1] = PR[GP1:90,1] + 14.064;
   1:  PR[GP1:91,2] = PR[GP1:90,2] + 22.133;
   1:L PR[91] R[100]mm/sec CNT100;
   1:  PR[GP1:91,1] = PR[GP1:90,1] + 9.100;
   1:  PR[GP1:91,2] = PR[GP1:90,2] + 22.930;
   1:L PR[91] R[100]mm/sec CNT100;
   1:  PR[GP1:91,1] = PR[GP1:90,1] + 7.911;
   1:  PR[GP1:91,2] = PR[GP1:90,2] + 23.086;
   1:L PR[91] R[100]mm/sec CNT100;
   1:  PR[GP1:91,1] = PR[GP1:90,1] + 2.523;
   1:  PR[GP1:91,2] = PR[GP1:90,2] + 22.566;
   1:L PR[91] R[100]mm/sec CNT100;
   1:  PR[GP1:91,1] = PR[GP1:90,1] + 1.655;
   1:  PR[GP1:91,2] = PR[GP1:90,2] + 22.457;
   1:L PR[91] R[100]mm/sec CNT100;
   1:  PR[GP1:91,1] = PR[GP1:90,1] + 0.733;
   1:  PR[GP1:91,2] = PR[GP1:90,2] + 22.162;
   1:L PR[91] R[100]mm/sec CNT100;
   1:  PR[91] = PR[90];
   1:  PR[GP1:91,1] = PR[GP1:90,1] + -0.559;
   1:  PR[GP1:91,2] = PR[GP1:90,2] + 22.331;
   1:  PR[GP1:91,3] = PR[GP1:90,3] + 55.815;
   1:L PR[91] R[100]mm/sec CNT100;
   1:  PR[GP1:91,1] = PR[GP1:90,1] + -1.280;
   1:  PR[GP1:91,2] = PR[GP1:90,2] + 22.562;
   1:L PR[91] R[100]mm/sec CNT100;
   1:  PR[GP1:91,1] = PR[GP1:90,1] + -1.902;
   1:  PR[GP1:91,2] = PR[GP1:90,2] + 22.640;
   1:L PR[91] R[100]mm/sec CNT100;
   1:  PR[GP1:91,1] = PR[GP1:90,1] + -7.554;
   1:  PR[GP1:91,2] = PR[GP1:90,2] + 23.185;
   1:L PR[91] R[100]mm/sec CNT100;
   1:  PR[GP1:91,1] = PR[GP1:90,1] + -8.493;
   1:  PR[GP1:91,2] = PR[GP1:90,2] + 23.062;
   1:L PR[91] R[100]mm/sec CNT100;
   1:  PR[GP1:91,1] = PR[GP1:90,1] + -13.722;
   1:  PR[GP1:91,2] = PR[GP1:90,2] + 22.224;
   1:L PR[91] R[100]mm/sec CNT100;
   1:  PR[GP1:91,1] = PR[GP1:90,1] + -14.845;
   1:  PR[GP1:91,2] = PR[GP1:90,2] + 21.769;
   1:L PR[91] R[100]mm/sec CNT100;
   1:  PR[GP1:91,1] = PR[GP1:90,1] + -19.428;
   1:  PR[GP1:91,2] = PR[GP1:90,2] + 19.770;
   1:L PR[91] R[100]mm/sec CNT100;
   1:  PR[GP1:91,1] = PR[GP1:90,1] + -20.591;
   1:  PR[GP1:91,2] = PR[GP1:90,2] + 18.905;
   1:L PR[91] R[100]mm/sec CNT100;
   1:  PR[GP1:91,1] = PR[GP1:90,1] + -24.292;
   1:  PR[GP1:91,2] = PR[GP1:90,2] + 16.006;
   1:L PR[91] R[100]mm/sec CNT100;
   1:  PR[GP1:91,1] = PR[GP1:90,1] + -25.312;
   1:  PR[GP1:91,2] = PR[GP1:90,2] + 14.717;
   1:L PR[91] R[100]mm/sec CNT100;
   1:  PR[GP1:91,1] = PR[GP1:90,1] + -28.004;
   1:  PR[GP1:91,2] = PR[GP1:90,2] + 11.174;
   1:L PR[91] R[100]mm/sec CNT100;
   1:  PR[GP1:91,1] = PR[GP1:90,1] + -28.704;
   1:  PR[GP1:91,2] = PR[GP1:90,2] + 9.555;
   1:L PR[91] R[100]mm/sec CNT100;
   1:  PR[GP1:91,1] = PR[GP1:90,1] + -30.325;
   1:  PR[GP1:91,2] = PR[GP1:90,2] + 5.637;
   1:L PR[91] R[100]mm/sec CNT100;
   1:  PR[GP1:91,1] = PR[GP1:90,1] + -30.572;
   1:  PR[GP1:91,2] = PR[GP1:90,2] + 3.813;
   1:L PR[91] R[100]mm/sec CNT100;
   1:  PR[GP1:91,1] = PR[GP1:90,1] + -30.817;
   1:  PR[GP1:91,2] = PR[GP1:90,2] + 1.344;
   1:L PR[91] R[100]mm/sec CNT100;
   1:  PR[GP1:91,1] = PR[GP1:90,1] + -31.038;
   1:  PR[GP1:91,2] = PR[GP1:90,2] + -0.338;
   1:L PR[91] R[100]mm/sec CNT100;
   1:  PR[GP1:91,1] = PR[GP1:90,1] + -30.861;
   1:  PR[GP1:91,2] = PR[GP1:90,2] + -2.182;
   1:L PR[91] R[100]mm/sec CNT100;
   1:  PR[GP1:91,1] = PR[GP1:90,1] + -30.322;
   1:  PR[GP1:91,2] = PR[GP1:90,2] + -6.270;
   1:L PR[91] R[100]mm/sec CNT100;
   1:  PR[GP1:91,1] = PR[GP1:90,1] + -28.699;
   1:  PR[GP1:91,2] = PR[GP1:90,2] + -10.189;
   1:L PR[91] R[100]mm/sec CNT100;
   1:  PR[GP1:91,1] = PR[GP1:90,1] + -27.998;
   1:  PR[GP1:91,2] = PR[GP1:90,2] + -11.808;
   1:L PR[91] R[100]mm/sec CNT100;
   1:  PR[GP1:91,1] = PR[GP1:90,1] + -25.301;
   1:  PR[GP1:91,2] = PR[GP1:90,2] + -15.354;
   1:L PR[91] R[100]mm/sec CNT100;
   1:  PR[GP1:91,1] = PR[GP1:90,1] + -24.278;
   1:  PR[GP1:91,2] = PR[GP1:90,2] + -16.644;
   1:L PR[91] R[100]mm/sec CNT100;
   1:  PR[GP1:91,1] = PR[GP1:90,1] + -20.571;
   1:  PR[GP1:91,2] = PR[GP1:90,2] + -19.543;
   1:L PR[91] R[100]mm/sec CNT100;
   1:  PR[GP1:91,1] = PR[GP1:90,1] + -19.406;
   1:  PR[GP1:91,2] = PR[GP1:90,2] + -20.407;
   1:L PR[91] R[100]mm/sec CNT100;
   1:  PR[GP1:91,1] = PR[GP1:90,1] + -14.816;
   1:  PR[GP1:91,2] = PR[GP1:90,2] + -22.403;
   1:L PR[91] R[100]mm/sec CNT100;
   1:  PR[GP1:91,1] = PR[GP1:90,1] + -13.692;
   1:  PR[GP1:91,2] = PR[GP1:90,2] + -22.857;
   1:L PR[91] R[100]mm/sec CNT100;
   1:  PR[GP1:91,1] = PR[GP1:90,1] + -8.456;
   1:  PR[GP1:91,2] = PR[GP1:90,2] + -23.689;
   1:L PR[91] R[100]mm/sec CNT100;
   1:  PR[GP1:91,1] = PR[GP1:90,1] + -7.518;
   1:  PR[GP1:91,2] = PR[GP1:90,2] + -23.810;
   1:L PR[91] R[100]mm/sec CNT100;
   1:  PR[GP1:91,1] = PR[GP1:90,1] + -1.809;
   1:  PR[GP1:91,2] = PR[GP1:90,2] + -23.245;
   1:L PR[91] R[100]mm/sec CNT100;
   1:  PR[GP1:91,1] = PR[GP1:90,1] + -1.233;
   1:  PR[GP1:91,2] = PR[GP1:90,2] + -23.172;
   1:L PR[91] R[100]mm/sec CNT100;
   1:  PR[GP1:91,1] = PR[GP1:90,1] + -0.557;
   1:  PR[GP1:91,2] = PR[GP1:90,2] + -22.957;
   1:L PR[91] R[100]mm/sec CNT100;
   1:  PR[GP1:91,1] = PR[GP1:90,1] + 0.645;
   1:  PR[GP1:91,2] = PR[GP1:90,2] + -22.959;
   1:L PR[91] R[100]mm/sec CNT100;
   1:  PR[GP1:91,1] = PR[GP1:90,1] + 2.026;
   1:  PR[GP1:91,2] = PR[GP1:90,2] + -23.252;
   1:L PR[91] R[100]mm/sec CNT100;
   1:  PR[GP1:91,1] = PR[GP1:90,1] + 7.676;
   1:  PR[GP1:91,2] = PR[GP1:90,2] + -23.810;
   1:L PR[91] R[100]mm/sec CNT100;
   1:  PR[GP1:91,1] = PR[GP1:90,1] + 8.614;
   1:  PR[GP1:91,2] = PR[GP1:90,2] + -23.689;
   1:L PR[91] R[100]mm/sec CNT100;
   1:  PR[GP1:91,1] = PR[GP1:90,1] + 13.850;
   1:  PR[GP1:91,2] = PR[GP1:90,2] + -22.856;
   1:L PR[91] R[100]mm/sec CNT100;
   1:  PR[GP1:91,1] = PR[GP1:90,1] + 14.974;
   1:  PR[GP1:91,2] = PR[GP1:90,2] + -22.403;
   1:L PR[91] R[100]mm/sec CNT100;
   1:  PR[GP1:91,1] = PR[GP1:90,1] + 19.563;
   1:  PR[GP1:91,2] = PR[GP1:90,2] + -20.407;
   1:L PR[91] R[100]mm/sec CNT100;
   1:  PR[GP1:91,1] = PR[GP1:90,1] + 20.729;
   1:  PR[GP1:91,2] = PR[GP1:90,2] + -19.543;
   1:L PR[91] R[100]mm/sec CNT100;
   1:  PR[GP1:91,1] = PR[GP1:90,1] + 24.435;
   1:  PR[GP1:91,2] = PR[GP1:90,2] + -16.644;
   1:L PR[91] R[100]mm/sec CNT100;
   1:  PR[GP1:91,1] = PR[GP1:90,1] + 25.458;
   1:  PR[GP1:91,2] = PR[GP1:90,2] + -15.352;
   1:L PR[91] R[100]mm/sec CNT100;
   1:  PR[GP1:91,1] = PR[GP1:90,1] + 28.155;
   1:  PR[GP1:91,2] = PR[GP1:90,2] + -11.803;
   1:L PR[91] R[100]mm/sec CNT100;
   1:  PR[GP1:91,1] = PR[GP1:90,1] + 28.856;
   1:  PR[GP1:91,2] = PR[GP1:90,2] + -10.191;
   1:L PR[91] R[100]mm/sec CNT100;
   1:  PR[GP1:91,1] = PR[GP1:90,1] + 30.480;
   1:  PR[GP1:91,2] = PR[GP1:90,2] + -6.276;
   1:L PR[91] R[100]mm/sec CNT100;
   1:  PR[GP1:91,1] = PR[GP1:90,1] + 30.728;
   1:  PR[GP1:91,2] = PR[GP1:90,2] + -4.444;
   1:L PR[91] R[100]mm/sec CNT100;
   1:  PR[GP1:91,1] = PR[GP1:90,1] + 30.973;
   1:  PR[GP1:91,2] = PR[GP1:90,2] + -1.971;
   1:L PR[91] R[100]mm/sec CNT100;
   1:  PR[GP1:91,1] = PR[GP1:90,1] + 31.195;
   1:  PR[GP1:91,2] = PR[GP1:90,2] + -0.286;
   1:L PR[91] R[100]mm/sec CNT100;
   1:  PR[GP1:91,1] = PR[GP1:90,1] + 31.019;
   1:  PR[GP1:91,2] = PR[GP1:90,2] + 1.562;
   1:L PR[91] R[100]mm/sec CNT100;
   1:  PR[GP1:91,1] = PR[GP1:90,1] + 30.481;
   1:  PR[GP1:91,2] = PR[GP1:90,2] + 5.649;
   1:L PR[91] R[100]mm/sec CNT100;
   1:  PR[GP1:91,1] = PR[GP1:90,1] + 28.861;
   1:  PR[GP1:91,2] = PR[GP1:90,2] + 9.558;
   1:L PR[91] R[100]mm/sec CNT100;
   1:  PR[GP1:91,1] = PR[GP1:90,1] + 28.161;
   1:  PR[GP1:91,2] = PR[GP1:90,2] + 11.169;
   1:L PR[91] R[100]mm/sec CNT100;
   1:  PR[GP1:91,1] = PR[GP1:90,1] + 25.469;
   1:  PR[GP1:91,2] = PR[GP1:90,2] + 14.715;
   1:L PR[91] R[100]mm/sec CNT100;
   1:  PR[GP1:91,1] = PR[GP1:90,1] + 24.448;
   1:  PR[GP1:91,2] = PR[GP1:90,2] + 16.007;
   1:L PR[91] R[100]mm/sec CNT100;
   1:  PR[GP1:91,1] = PR[GP1:90,1] + 20.748;
   1:  PR[GP1:91,2] = PR[GP1:90,2] + 18.906;
   1:L PR[91] R[100]mm/sec CNT100;
   1:  PR[GP1:91,1] = PR[GP1:90,1] + 19.585;
   1:  PR[GP1:91,2] = PR[GP1:90,2] + 19.770;
   1:L PR[91] R[100]mm/sec CNT100;
   1:  PR[GP1:91,1] = PR[GP1:90,1] + 15.003;
   1:  PR[GP1:91,2] = PR[GP1:90,2] + 21.769;
   1:L PR[91] R[100]mm/sec CNT100;
   1:  PR[GP1:91,1] = PR[GP1:90,1] + 13.879;
   1:  PR[GP1:91,2] = PR[GP1:90,2] + 22.223;
   1:L PR[91] R[100]mm/sec CNT100;
   1:  PR[GP1:91,1] = PR[GP1:90,1] + 8.651;
   1:  PR[GP1:91,2] = PR[GP1:90,2] + 23.062;
   1:L PR[91] R[100]mm/sec CNT100;
   1:  PR[GP1:91,1] = PR[GP1:90,1] + 7.712;
   1:  PR[GP1:91,2] = PR[GP1:90,2] + 23.185;
   1:L PR[91] R[100]mm/sec CNT100;
   1:  PR[GP1:91,1] = PR[GP1:90,1] + 2.060;
   1:  PR[GP1:91,2] = PR[GP1:90,2] + 22.640;
   1:L PR[91] R[100]mm/sec CNT100;
   1:  PR[GP1:91,1] = PR[GP1:90,1] + 1.439;
   1:  PR[GP1:91,2] = PR[GP1:90,2] + 22.562;
   1:L PR[91] R[100]mm/sec CNT100;
   1:  PR[GP1:91,1] = PR[GP1:90,1] + 0.718;
   1:  PR[GP1:91,2] = PR[GP1:90,2] + 22.331;
   1:L PR[91] R[100]mm/sec CNT100;
   1:  PR[91] = PR[90];
   1:  PR[GP1:91,1] = PR[GP1:90,1] + -0.544;
   1:  PR[GP1:91,2] = PR[GP1:90,2] + 22.501;
   1:  PR[GP1:91,3] = PR[GP1:90,3] + 56.425;
   1:L PR[91] R[100]mm/sec CNT100;
   1:  PR[GP1:91,1] = PR[GP1:90,1] + -1.064;
   1:  PR[GP1:91,2] = PR[GP1:90,2] + 22.667;
   1:L PR[91] R[100]mm/sec CNT100;
   1:  PR[GP1:91,1] = PR[GP1:90,1] + -1.438;
   1:  PR[GP1:91,2] = PR[GP1:90,2] + 22.714;
   1:L PR[91] R[100]mm/sec CNT100;
   1:  PR[GP1:91,1] = PR[GP1:90,1] + -7.355;
   1:  PR[GP1:91,2] = PR[GP1:90,2] + 23.285;
   1:L PR[91] R[100]mm/sec CNT100;
   1:  PR[GP1:91,1] = PR[GP1:90,1] + -8.043;
   1:  PR[GP1:91,2] = PR[GP1:90,2] + 23.194;
   1:L PR[91] R[100]mm/sec CNT100;
   1:  PR[GP1:91,1] = PR[GP1:90,1] + -13.537;
   1:  PR[GP1:91,2] = PR[GP1:90,2] + 22.314;
   1:L PR[91] R[100]mm/sec CNT100;
   1:  PR[GP1:91,1] = PR[GP1:90,1] + -14.421;
   1:  PR[GP1:91,2] = PR[GP1:90,2] + 21.956;
   1:L PR[91] R[100]mm/sec CNT100;
   1:  PR[GP1:91,1] = PR[GP1:90,1] + -19.255;
   1:  PR[GP1:91,2] = PR[GP1:90,2] + 19.847;
   1:L PR[91] R[100]mm/sec CNT100;
   1:  PR[GP1:91,1] = PR[GP1:90,1] + -20.209;
   1:  PR[GP1:91,2] = PR[GP1:90,2] + 19.139;
   1:L PR[91] R[100]mm/sec CNT100;
   1:  PR[GP1:91,1] = PR[GP1:90,1] + -24.129;
   1:  PR[GP1:91,2] = PR[GP1:90,2] + 16.067;
   1:L PR[91] R[100]mm/sec CNT100;
   1:  PR[GP1:91,1] = PR[GP1:90,1] + -24.986;
   1:  PR[GP1:91,2] = PR[GP1:90,2] + 14.984;
   1:L PR[91] R[100]mm/sec CNT100;
   1:  PR[GP1:91,1] = PR[GP1:90,1] + -27.849;
   1:  PR[GP1:91,2] = PR[GP1:90,2] + 11.216;
   1:L PR[91] R[100]mm/sec CNT100;
   1:  PR[GP1:91,1] = PR[GP1:90,1] + -28.445;
   1:  PR[GP1:91,2] = PR[GP1:90,2] + 9.837;
   1:L PR[91] R[100]mm/sec CNT100;
   1:  PR[GP1:91,1] = PR[GP1:90,1] + -30.175;
   1:  PR[GP1:91,2] = PR[GP1:90,2] + 5.659;
   1:L PR[91] R[100]mm/sec CNT100;
   1:  PR[GP1:91,1] = PR[GP1:90,1] + -30.387;
   1:  PR[GP1:91,2] = PR[GP1:90,2] + 4.093;
   1:L PR[91] R[100]mm/sec CNT100;
   1:  PR[GP1:91,1] = PR[GP1:90,1] + -30.600;
   1:  PR[GP1:91,2] = PR[GP1:90,2] + 1.940;
   1:L PR[91] R[100]mm/sec CNT100;
   1:  PR[GP1:91,1] = PR[GP1:90,1] + -30.899;
   1:  PR[GP1:91,2] = PR[GP1:90,2] + -0.338;
   1:L PR[91] R[100]mm/sec CNT100;
   1:  PR[GP1:91,1] = PR[GP1:90,1] + -30.747;
   1:  PR[GP1:91,2] = PR[GP1:90,2] + -1.930;
   1:L PR[91] R[100]mm/sec CNT100;
   1:  PR[GP1:91,1] = PR[GP1:90,1] + -30.172;
   1:  PR[GP1:91,2] = PR[GP1:90,2] + -6.291;
   1:L PR[91] R[100]mm/sec CNT100;
   1:  PR[GP1:91,1] = PR[GP1:90,1] + -28.440;
   1:  PR[GP1:91,2] = PR[GP1:90,2] + -10.470;
   1:L PR[91] R[100]mm/sec CNT100;
   1:  PR[GP1:91,1] = PR[GP1:90,1] + -27.843;
   1:  PR[GP1:91,2] = PR[GP1:90,2] + -11.851;
   1:L PR[91] R[100]mm/sec CNT100;
   1:  PR[GP1:91,1] = PR[GP1:90,1] + -24.975;
   1:  PR[GP1:91,2] = PR[GP1:90,2] + -15.621;
   1:L PR[91] R[100]mm/sec CNT100;
   1:  PR[GP1:91,1] = PR[GP1:90,1] + -24.116;
   1:  PR[GP1:91,2] = PR[GP1:90,2] + -16.704;
   1:L PR[91] R[100]mm/sec CNT100;
   1:  PR[GP1:91,1] = PR[GP1:90,1] + -20.188;
   1:  PR[GP1:91,2] = PR[GP1:90,2] + -19.776;
   1:L PR[91] R[100]mm/sec CNT100;
   1:  PR[GP1:91,1] = PR[GP1:90,1] + -19.234;
   1:  PR[GP1:91,2] = PR[GP1:90,2] + -20.484;
   1:L PR[91] R[100]mm/sec CNT100;
   1:  PR[GP1:91,1] = PR[GP1:90,1] + -14.392;
   1:  PR[GP1:91,2] = PR[GP1:90,2] + -22.590;
   1:L PR[91] R[100]mm/sec CNT100;
   1:  PR[GP1:91,1] = PR[GP1:90,1] + -13.508;
   1:  PR[GP1:91,2] = PR[GP1:90,2] + -22.947;
   1:L PR[91] R[100]mm/sec CNT100;
   1:  PR[GP1:91,1] = PR[GP1:90,1] + -8.006;
   1:  PR[GP1:91,2] = PR[GP1:90,2] + -23.821;
   1:L PR[91] R[100]mm/sec CNT100;
   1:  PR[GP1:91,1] = PR[GP1:90,1] + -7.319;
   1:  PR[GP1:91,2] = PR[GP1:90,2] + -23.910;
   1:L PR[91] R[100]mm/sec CNT100;
   1:  PR[GP1:91,1] = PR[GP1:90,1] + -1.344;
   1:  PR[GP1:91,2] = PR[GP1:90,2] + -23.319;
   1:L PR[91] R[100]mm/sec CNT100;
   1:  PR[GP1:91,1] = PR[GP1:90,1] + -1.015;
   1:  PR[GP1:91,2] = PR[GP1:90,2] + -23.277;
   1:L PR[91] R[100]mm/sec CNT100;
   1:  PR[GP1:91,1] = PR[GP1:90,1] + -0.540;
   1:  PR[GP1:91,2] = PR[GP1:90,2] + -23.127;
   1:L PR[91] R[100]mm/sec CNT100;
   1:  PR[GP1:91,1] = PR[GP1:90,1] + 0.629;
   1:L PR[91] R[100]mm/sec CNT100;
   1:  PR[GP1:91,1] = PR[GP1:90,1] + 1.561;
   1:  PR[GP1:91,2] = PR[GP1:90,2] + -23.325;
   1:L PR[91] R[100]mm/sec CNT100;
   1:  PR[GP1:91,1] = PR[GP1:90,1] + 7.477;
   1:  PR[GP1:91,2] = PR[GP1:90,2] + -23.910;
   1:L PR[91] R[100]mm/sec CNT100;
   1:  PR[GP1:91,1] = PR[GP1:90,1] + 8.164;
   1:  PR[GP1:91,2] = PR[GP1:90,2] + -23.821;
   1:L PR[91] R[100]mm/sec CNT100;
   1:  PR[GP1:91,1] = PR[GP1:90,1] + 13.666;
   1:  PR[GP1:91,2] = PR[GP1:90,2] + -22.946;
   1:L PR[91] R[100]mm/sec CNT100;
   1:  PR[GP1:91,1] = PR[GP1:90,1] + 14.550;
   1:  PR[GP1:91,2] = PR[GP1:90,2] + -22.590;
   1:L PR[91] R[100]mm/sec CNT100;
   1:  PR[GP1:91,1] = PR[GP1:90,1] + 19.392;
   1:  PR[GP1:91,2] = PR[GP1:90,2] + -20.484;
   1:L PR[91] R[100]mm/sec CNT100;
   1:  PR[GP1:91,1] = PR[GP1:90,1] + 20.346;
   1:  PR[GP1:91,2] = PR[GP1:90,2] + -19.776;
   1:L PR[91] R[100]mm/sec CNT100;
   1:  PR[GP1:91,1] = PR[GP1:90,1] + 24.273;
   1:  PR[GP1:91,2] = PR[GP1:90,2] + -16.705;
   1:L PR[91] R[100]mm/sec CNT100;
   1:  PR[GP1:91,1] = PR[GP1:90,1] + 25.132;
   1:  PR[GP1:91,2] = PR[GP1:90,2] + -15.619;
   1:L PR[91] R[100]mm/sec CNT100;
   1:  PR[GP1:91,1] = PR[GP1:90,1] + 28.000;
   1:  PR[GP1:91,2] = PR[GP1:90,2] + -11.846;
   1:L PR[91] R[100]mm/sec CNT100;
   1:  PR[GP1:91,1] = PR[GP1:90,1] + 28.598;
   1:  PR[GP1:91,2] = PR[GP1:90,2] + -10.471;
   1:L PR[91] R[100]mm/sec CNT100;
   1:  PR[GP1:91,1] = PR[GP1:90,1] + 30.330;
   1:  PR[GP1:91,2] = PR[GP1:90,2] + -6.297;
   1:L PR[91] R[100]mm/sec CNT100;
   1:  PR[GP1:91,1] = PR[GP1:90,1] + 30.542;
   1:  PR[GP1:91,2] = PR[GP1:90,2] + -4.725;
   1:L PR[91] R[100]mm/sec CNT100;
   1:  PR[GP1:91,1] = PR[GP1:90,1] + 30.756;
   1:  PR[GP1:91,2] = PR[GP1:90,2] + -2.568;
   1:L PR[91] R[100]mm/sec CNT100;
   1:  PR[GP1:91,1] = PR[GP1:90,1] + 31.056;
   1:  PR[GP1:91,2] = PR[GP1:90,2] + -0.286;
   1:L PR[91] R[100]mm/sec CNT100;
   1:  PR[GP1:91,1] = PR[GP1:90,1] + 30.904;
   1:  PR[GP1:91,2] = PR[GP1:90,2] + 1.310;
   1:L PR[91] R[100]mm/sec CNT100;
   1:  PR[GP1:91,1] = PR[GP1:90,1] + 30.330;
   1:  PR[GP1:91,2] = PR[GP1:90,2] + 5.670;
   1:L PR[91] R[100]mm/sec CNT100;
   1:  PR[GP1:91,1] = PR[GP1:90,1] + 28.603;
   1:  PR[GP1:91,2] = PR[GP1:90,2] + 9.838;
   1:L PR[91] R[100]mm/sec CNT100;
   1:  PR[GP1:91,1] = PR[GP1:90,1] + 28.006;
   1:  PR[GP1:91,2] = PR[GP1:90,2] + 11.211;
   1:L PR[91] R[100]mm/sec CNT100;
   1:  PR[GP1:91,1] = PR[GP1:90,1] + 25.143;
   1:  PR[GP1:91,2] = PR[GP1:90,2] + 14.983;
   1:L PR[91] R[100]mm/sec CNT100;
   1:  PR[GP1:91,1] = PR[GP1:90,1] + 24.286;
   1:  PR[GP1:91,2] = PR[GP1:90,2] + 16.068;
   1:L PR[91] R[100]mm/sec CNT100;
   1:  PR[GP1:91,1] = PR[GP1:90,1] + 20.366;
   1:  PR[GP1:91,2] = PR[GP1:90,2] + 19.139;
   1:L PR[91] R[100]mm/sec CNT100;
   1:  PR[GP1:91,1] = PR[GP1:90,1] + 19.413;
   1:  PR[GP1:91,2] = PR[GP1:90,2] + 19.847;
   1:L PR[91] R[100]mm/sec CNT100;
   1:  PR[GP1:91,1] = PR[GP1:90,1] + 14.579;
   1:  PR[GP1:91,2] = PR[GP1:90,2] + 21.956;
   1:L PR[91] R[100]mm/sec CNT100;
   1:  PR[GP1:91,1] = PR[GP1:90,1] + 13.695;
   1:  PR[GP1:91,2] = PR[GP1:90,2] + 22.313;
   1:L PR[91] R[100]mm/sec CNT100;
   1:  PR[GP1:91,1] = PR[GP1:90,1] + 8.201;
   1:  PR[GP1:91,2] = PR[GP1:90,2] + 23.194;
   1:L PR[91] R[100]mm/sec CNT100;
   1:  PR[GP1:91,1] = PR[GP1:90,1] + 7.513;
   1:  PR[GP1:91,2] = PR[GP1:90,2] + 23.285;
   1:L PR[91] R[100]mm/sec CNT100;
   1:  PR[GP1:91,1] = PR[GP1:90,1] + 1.597;
   1:  PR[GP1:91,2] = PR[GP1:90,2] + 22.714;
   1:L PR[91] R[100]mm/sec CNT100;
   1:  PR[GP1:91,1] = PR[GP1:90,1] + 1.222;
   1:  PR[GP1:91,2] = PR[GP1:90,2] + 22.667;
   1:L PR[91] R[100]mm/sec CNT100;
   1:  PR[GP1:91,1] = PR[GP1:90,1] + 0.703;
   1:  PR[GP1:91,2] = PR[GP1:90,2] + 22.501;
   1:L PR[91] R[100]mm/sec CNT100;
   1:  PR[91] = PR[90];
   1:  PR[GP1:91,1] = PR[GP1:90,1] + -0.529;
   1:  PR[GP1:91,2] = PR[GP1:90,2] + 22.670;
   1:  PR[GP1:91,3] = PR[GP1:90,3] + 57.035;
   1:L PR[91] R[100]mm/sec CNT100;
   1:  PR[GP1:91,1] = PR[GP1:90,1] + -0.847;
   1:  PR[GP1:91,2] = PR[GP1:90,2] + 22.772;
   1:L PR[91] R[100]mm/sec CNT100;
   1:  PR[GP1:91,1] = PR[GP1:90,1] + -0.976;
   1:  PR[GP1:91,2] = PR[GP1:90,2] + 22.788;
   1:L PR[91] R[100]mm/sec CNT100;
   1:  PR[GP1:91,1] = PR[GP1:90,1] + -7.156;
   1:  PR[GP1:91,2] = PR[GP1:90,2] + 23.384;
   1:L PR[91] R[100]mm/sec CNT100;
   1:  PR[GP1:91,1] = PR[GP1:90,1] + -7.594;
   1:  PR[GP1:91,2] = PR[GP1:90,2] + 23.327;
   1:L PR[91] R[100]mm/sec CNT100;
   1:  PR[GP1:91,1] = PR[GP1:90,1] + -13.353;
   1:  PR[GP1:91,2] = PR[GP1:90,2] + 22.404;
   1:L PR[91] R[100]mm/sec CNT100;
   1:  PR[GP1:91,1] = PR[GP1:90,1] + -13.996;
   1:  PR[GP1:91,2] = PR[GP1:90,2] + 22.143;
   1:L PR[91] R[100]mm/sec CNT100;
   1:  PR[GP1:91,1] = PR[GP1:90,1] + -19.083;
   1:  PR[GP1:91,2] = PR[GP1:90,2] + 19.924;
   1:L PR[91] R[100]mm/sec CNT100;
   1:  PR[GP1:91,1] = PR[GP1:90,1] + -19.826;
   1:  PR[GP1:91,2] = PR[GP1:90,2] + 19.372;
   1:L PR[91] R[100]mm/sec CNT100;
   1:  PR[GP1:91,1] = PR[GP1:90,1] + -23.967;
   1:  PR[GP1:91,2] = PR[GP1:90,2] + 16.128;
   1:L PR[91] R[100]mm/sec CNT100;
   1:  PR[GP1:91,1] = PR[GP1:90,1] + -24.660;
   1:  PR[GP1:91,2] = PR[GP1:90,2] + 15.252;
   1:L PR[91] R[100]mm/sec CNT100;
   1:  PR[GP1:91,1] = PR[GP1:90,1] + -27.694;
   1:  PR[GP1:91,2] = PR[GP1:90,2] + 11.258;
   1:L PR[91] R[100]mm/sec CNT100;
   1:  PR[GP1:91,1] = PR[GP1:90,1] + -28.187;
   1:  PR[GP1:91,2] = PR[GP1:90,2] + 10.118;
   1:L PR[91] R[100]mm/sec CNT100;
   1:  PR[GP1:91,1] = PR[GP1:90,1] + -30.024;
   1:  PR[GP1:91,2] = PR[GP1:90,2] + 5.680;
   1:L PR[91] R[100]mm/sec CNT100;
   1:  PR[GP1:91,1] = PR[GP1:90,1] + -30.201;
   1:  PR[GP1:91,2] = PR[GP1:90,2] + 4.374;
   1:L PR[91] R[100]mm/sec CNT100;
   1:  PR[GP1:91,1] = PR[GP1:90,1] + -30.383;
   1:  PR[GP1:91,2] = PR[GP1:90,2] + 2.537;
   1:L PR[91] R[100]mm/sec CNT100;
   1:  PR[GP1:91,1] = PR[GP1:90,1] + -30.761;
   1:  PR[GP1:91,2] = PR[GP1:90,2] + -0.338;
   1:L PR[91] R[100]mm/sec CNT100;
   1:  PR[GP1:91,1] = PR[GP1:90,1] + -30.632;
   1:  PR[GP1:91,2] = PR[GP1:90,2] + -1.679;
   1:L PR[91] R[100]mm/sec CNT100;
   1:  PR[GP1:91,1] = PR[GP1:90,1] + -30.021;
   1:  PR[GP1:91,2] = PR[GP1:90,2] + -6.312;
   1:L PR[91] R[100]mm/sec CNT100;
   1:  PR[GP1:91,1] = PR[GP1:90,1] + -28.182;
   1:  PR[GP1:91,2] = PR[GP1:90,2] + -10.752;
   1:L PR[91] R[100]mm/sec CNT100;
   1:  PR[GP1:91,1] = PR[GP1:90,1] + -27.688;
   1:  PR[GP1:91,2] = PR[GP1:90,2] + -11.893;
   1:L PR[91] R[100]mm/sec CNT100;
   1:  PR[GP1:91,1] = PR[GP1:90,1] + -24.649;
   1:  PR[GP1:91,2] = PR[GP1:90,2] + -15.889;
   1:L PR[91] R[100]mm/sec CNT100;
   1:  PR[GP1:91,1] = PR[GP1:90,1] + -23.954;
   1:  PR[GP1:91,2] = PR[GP1:90,2] + -16.765;
   1:L PR[91] R[100]mm/sec CNT100;
   1:  PR[GP1:91,1] = PR[GP1:90,1] + -19.805;
   1:  PR[GP1:91,2] = PR[GP1:90,2] + -20.009;
   1:L PR[91] R[100]mm/sec CNT100;
   1:  PR[GP1:91,1] = PR[GP1:90,1] + -19.062;
   1:  PR[GP1:91,2] = PR[GP1:90,2] + -20.560;
   1:L PR[91] R[100]mm/sec CNT100;
   1:  PR[GP1:91,1] = PR[GP1:90,1] + -13.967;
   1:  PR[GP1:91,2] = PR[GP1:90,2] + -22.777;
   1:L PR[91] R[100]mm/sec CNT100;
   1:  PR[GP1:91,1] = PR[GP1:90,1] + -13.323;
   1:  PR[GP1:91,2] = PR[GP1:90,2] + -23.036;
   1:L PR[91] R[100]mm/sec CNT100;
   1:  PR[GP1:91,1] = PR[GP1:90,1] + -7.557;
   1:  PR[GP1:91,2] = PR[GP1:90,2] + -23.953;
   1:L PR[91] R[100]mm/sec CNT100;
   1:  PR[GP1:91,1] = PR[GP1:90,1] + -7.120;
   1:  PR[GP1:91,2] = PR[GP1:90,2] + -24.009;
   1:L PR[91] R[100]mm/sec CNT100;
   1:  PR[GP1:91,1] = PR[GP1:90,1] + -0.879;
   1:  PR[GP1:91,2] = PR[GP1:90,2] + -23.392;
   1:L PR[91] R[100]mm/sec CNT100;
   1:  PR[GP1:91,1] = PR[GP1:90,1] + -0.799;
   1:  PR[GP1:91,2] = PR[GP1:90,2] + -23.382;
   1:L PR[91] R[100]mm/sec CNT100;
   1:  PR[GP1:91,1] = PR[GP1:90,1] + -0.525;
   1:  PR[GP1:91,2] = PR[GP1:90,2] + -23.296;
   1:L PR[91] R[100]mm/sec CNT100;
   1:  PR[GP1:91,1] = PR[GP1:90,1] + 0.614;
   1:L PR[91] R[100]mm/sec CNT100;
   1:  PR[GP1:91,1] = PR[GP1:90,1] + 1.097;
   1:  PR[GP1:91,2] = PR[GP1:90,2] + -23.398;
   1:L PR[91] R[100]mm/sec CNT100;
   1:  PR[GP1:91,1] = PR[GP1:90,1] + 7.278;
   1:  PR[GP1:91,2] = PR[GP1:90,2] + -24.009;
   1:L PR[91] R[100]mm/sec CNT100;
   1:  PR[GP1:91,1] = PR[GP1:90,1] + 7.716;
   1:  PR[GP1:91,2] = PR[GP1:90,2] + -23.953;
   1:L PR[91] R[100]mm/sec CNT100;
   1:  PR[GP1:91,1] = PR[GP1:90,1] + 13.481;
   1:  PR[GP1:91,2] = PR[GP1:90,2] + -23.036;
   1:L PR[91] R[100]mm/sec CNT100;
   1:  PR[GP1:91,1] = PR[GP1:90,1] + 14.126;
   1:  PR[GP1:91,2] = PR[GP1:90,2] + -22.776;
   1:L PR[91] R[100]mm/sec CNT100;
   1:  PR[GP1:91,1] = PR[GP1:90,1] + 19.220;
   1:  PR[GP1:91,2] = PR[GP1:90,2] + -20.561;
   1:L PR[91] R[100]mm/sec CNT100;
   1:  PR[GP1:91,1] = PR[GP1:90,1] + 19.963;
   1:  PR[GP1:91,2] = PR[GP1:90,2] + -20.009;
   1:L PR[91] R[100]mm/sec CNT100;
   1:  PR[GP1:91,1] = PR[GP1:90,1] + 24.111;
   1:  PR[GP1:91,2] = PR[GP1:90,2] + -16.765;
   1:L PR[91] R[100]mm/sec CNT100;
   1:  PR[GP1:91,1] = PR[GP1:90,1] + 24.806;
   1:  PR[GP1:91,2] = PR[GP1:90,2] + -15.887;
   1:L PR[91] R[100]mm/sec CNT100;
   1:  PR[GP1:91,1] = PR[GP1:90,1] + 27.845;
   1:  PR[GP1:91,2] = PR[GP1:90,2] + -11.889;
   1:L PR[91] R[100]mm/sec CNT100;
   1:  PR[GP1:91,1] = PR[GP1:90,1] + 28.340;
   1:  PR[GP1:91,2] = PR[GP1:90,2] + -10.752;
   1:L PR[91] R[100]mm/sec CNT100;
   1:  PR[GP1:91,1] = PR[GP1:90,1] + 30.179;
   1:  PR[GP1:91,2] = PR[GP1:90,2] + -6.318;
   1:L PR[91] R[100]mm/sec CNT100;
   1:  PR[GP1:91,1] = PR[GP1:90,1] + 30.357;
   1:  PR[GP1:91,2] = PR[GP1:90,2] + -5.007;
   1:L PR[91] R[100]mm/sec CNT100;
   1:  PR[GP1:91,1] = PR[GP1:90,1] + 30.539;
   1:  PR[GP1:91,2] = PR[GP1:90,2] + -3.166;
   1:L PR[91] R[100]mm/sec CNT100;
   1:  PR[GP1:91,1] = PR[GP1:90,1] + 30.918;
   1:  PR[GP1:91,2] = PR[GP1:90,2] + -0.286;
   1:L PR[91] R[100]mm/sec CNT100;
   1:  PR[GP1:91,1] = PR[GP1:90,1] + 30.790;
   1:  PR[GP1:91,2] = PR[GP1:90,2] + 1.057;
   1:L PR[91] R[100]mm/sec CNT100;
   1:  PR[GP1:91,1] = PR[GP1:90,1] + 30.180;
   1:  PR[GP1:91,2] = PR[GP1:90,2] + 5.690;
   1:L PR[91] R[100]mm/sec CNT100;
   1:  PR[GP1:91,1] = PR[GP1:90,1] + 28.344;
   1:  PR[GP1:91,2] = PR[GP1:90,2] + 10.118;
   1:L PR[91] R[100]mm/sec CNT100;
   1:  PR[GP1:91,1] = PR[GP1:90,1] + 27.851;
   1:  PR[GP1:91,2] = PR[GP1:90,2] + 11.254;
   1:L PR[91] R[100]mm/sec CNT100;
   1:  PR[GP1:91,1] = PR[GP1:90,1] + 24.817;
   1:  PR[GP1:91,2] = PR[GP1:90,2] + 15.251;
   1:L PR[91] R[100]mm/sec CNT100;
   1:  PR[GP1:91,1] = PR[GP1:90,1] + 24.123;
   1:  PR[GP1:91,2] = PR[GP1:90,2] + 16.128;
   1:L PR[91] R[100]mm/sec CNT100;
   1:  PR[GP1:91,1] = PR[GP1:90,1] + 19.983;
   1:  PR[GP1:91,2] = PR[GP1:90,2] + 19.372;
   1:L PR[91] R[100]mm/sec CNT100;
   1:  PR[GP1:91,1] = PR[GP1:90,1] + 19.241;
   1:  PR[GP1:91,2] = PR[GP1:90,2] + 19.924;
   1:L PR[91] R[100]mm/sec CNT100;
   1:  PR[GP1:91,1] = PR[GP1:90,1] + 14.154;
   1:  PR[GP1:91,2] = PR[GP1:90,2] + 22.143;
   1:L PR[91] R[100]mm/sec CNT100;
   1:  PR[GP1:91,1] = PR[GP1:90,1] + 13.511;
   1:  PR[GP1:91,2] = PR[GP1:90,2] + 22.403;
   1:L PR[91] R[100]mm/sec CNT100;
   1:  PR[GP1:91,1] = PR[GP1:90,1] + 7.752;
   1:  PR[GP1:91,2] = PR[GP1:90,2] + 23.327;
   1:L PR[91] R[100]mm/sec CNT100;
   1:  PR[GP1:91,1] = PR[GP1:90,1] + 7.314;
   1:  PR[GP1:91,2] = PR[GP1:90,2] + 23.384;
   1:L PR[91] R[100]mm/sec CNT100;
   1:  PR[GP1:91,1] = PR[GP1:90,1] + 1.135;
   1:  PR[GP1:91,2] = PR[GP1:90,2] + 22.788;
   1:L PR[91] R[100]mm/sec CNT100;
   1:  PR[GP1:91,1] = PR[GP1:90,1] + 1.006;
   1:  PR[GP1:91,2] = PR[GP1:90,2] + 22.772;
   1:L PR[91] R[100]mm/sec CNT100;
   1:  PR[GP1:91,1] = PR[GP1:90,1] + 0.688;
   1:  PR[GP1:91,2] = PR[GP1:90,2] + 22.670;
   1:L PR[91] R[100]mm/sec CNT100;
   1:  PR[91] = PR[90];
   1:  PR[GP1:91,1] = PR[GP1:90,1] + -0.359;
   1:  PR[GP1:91,2] = PR[GP1:90,2] + 22.840;
   1:  PR[GP1:91,3] = PR[GP1:90,3] + 57.645;
   1:L PR[91] R[100]mm/sec CNT100;
   1:  PR[GP1:91,1] = PR[GP1:90,1] + -6.957;
   1:  PR[GP1:91,2] = PR[GP1:90,2] + 23.484;
   1:L PR[91] R[100]mm/sec CNT100;
   1:  PR[GP1:91,1] = PR[GP1:90,1] + -7.145;
   1:  PR[GP1:91,2] = PR[GP1:90,2] + 23.459;
   1:L PR[91] R[100]mm/sec CNT100;
   1:  PR[GP1:91,1] = PR[GP1:90,1] + -13.168;
   1:  PR[GP1:91,2] = PR[GP1:90,2] + 22.494;
   1:L PR[91] R[100]mm/sec CNT100;
   1:  PR[GP1:91,1] = PR[GP1:90,1] + -13.572;
   1:  PR[GP1:91,2] = PR[GP1:90,2] + 22.330;
   1:L PR[91] R[100]mm/sec CNT100;
   1:  PR[GP1:91,1] = PR[GP1:90,1] + -18.911;
   1:  PR[GP1:91,2] = PR[GP1:90,2] + 20.001;
   1:L PR[91] R[100]mm/sec CNT100;
   1:  PR[GP1:91,1] = PR[GP1:90,1] + -19.443;
   1:  PR[GP1:91,2] = PR[GP1:90,2] + 19.605;
   1:L PR[91] R[100]mm/sec CNT100;
   1:  PR[GP1:91,1] = PR[GP1:90,1] + -23.805;
   1:  PR[GP1:91,2] = PR[GP1:90,2] + 16.189;
   1:L PR[91] R[100]mm/sec CNT100;
   1:  PR[GP1:91,1] = PR[GP1:90,1] + -24.335;
   1:  PR[GP1:91,2] = PR[GP1:90,2] + 15.519;
   1:L PR[91] R[100]mm/sec CNT100;
   1:  PR[GP1:91,1] = PR[GP1:90,1] + -27.539;
   1:  PR[GP1:91,2] = PR[GP1:90,2] + 11.301;
   1:L PR[91] R[100]mm/sec CNT100;
   1:  PR[GP1:91,1] = PR[GP1:90,1] + -27.929;
   1:  PR[GP1:91,2] = PR[GP1:90,2] + 10.399;
   1:L PR[91] R[100]mm/sec CNT100;
   1:  PR[GP1:91,1] = PR[GP1:90,1] + -29.874;
   1:  PR[GP1:91,2] = PR[GP1:90,2] + 5.701;
   1:L PR[91] R[100]mm/sec CNT100;
   1:  PR[GP1:91,1] = PR[GP1:90,1] + -30.015;
   1:  PR[GP1:91,2] = PR[GP1:90,2] + 4.655;
   1:L PR[91] R[100]mm/sec CNT100;
   1:  PR[GP1:91,1] = PR[GP1:90,1] + -30.166;
   1:  PR[GP1:91,2] = PR[GP1:90,2] + 3.133;
   1:L PR[91] R[100]mm/sec CNT100;
   1:  PR[GP1:91,1] = PR[GP1:90,1] + -30.622;
   1:  PR[GP1:91,2] = PR[GP1:90,2] + -0.338;
   1:L PR[91] R[100]mm/sec CNT100;
   1:  PR[GP1:91,1] = PR[GP1:90,1] + -30.518;
   1:  PR[GP1:91,2] = PR[GP1:90,2] + -1.427;
   1:L PR[91] R[100]mm/sec CNT100;
   1:  PR[GP1:91,1] = PR[GP1:90,1] + -29.871;
   1:  PR[GP1:91,2] = PR[GP1:90,2] + -6.333;
   1:L PR[91] R[100]mm/sec CNT100;
   1:  PR[GP1:91,1] = PR[GP1:90,1] + -27.923;
   1:  PR[GP1:91,2] = PR[GP1:90,2] + -11.033;
   1:L PR[91] R[100]mm/sec CNT100;
   1:  PR[GP1:91,1] = PR[GP1:90,1] + -27.533;
   1:  PR[GP1:91,2] = PR[GP1:90,2] + -11.936;
   1:L PR[91] R[100]mm/sec CNT100;
   1:  PR[GP1:91,1] = PR[GP1:90,1] + -24.323;
   1:  PR[GP1:91,2] = PR[GP1:90,2] + -16.156;
   1:L PR[91] R[100]mm/sec CNT100;
   1:  PR[GP1:91,1] = PR[GP1:90,1] + -23.792;
   1:  PR[GP1:91,2] = PR[GP1:90,2] + -16.826;
   1:L PR[91] R[100]mm/sec CNT100;
   1:  PR[GP1:91,1] = PR[GP1:90,1] + -19.423;
   1:  PR[GP1:91,2] = PR[GP1:90,2] + -20.242;
   1:L PR[91] R[100]mm/sec CNT100;
   1:  PR[GP1:91,1] = PR[GP1:90,1] + -18.890;
   1:  PR[GP1:91,2] = PR[GP1:90,2] + -20.637;
   1:L PR[91] R[100]mm/sec CNT100;
   1:  PR[GP1:91,1] = PR[GP1:90,1] + -13.543;
   1:  PR[GP1:91,2] = PR[GP1:90,2] + -22.964;
   1:L PR[91] R[100]mm/sec CNT100;
   1:  PR[GP1:91,1] = PR[GP1:90,1] + -13.139;
   1:  PR[GP1:91,2] = PR[GP1:90,2] + -23.126;
   1:L PR[91] R[100]mm/sec CNT100;
   1:  PR[GP1:91,1] = PR[GP1:90,1] + -7.108;
   1:  PR[GP1:91,2] = PR[GP1:90,2] + -24.085;
   1:L PR[91] R[100]mm/sec CNT100;
   1:  PR[GP1:91,1] = PR[GP1:90,1] + -6.921;
   1:  PR[GP1:91,2] = PR[GP1:90,2] + -24.109;
   1:L PR[91] R[100]mm/sec CNT100;
   1:  PR[GP1:91,1] = PR[GP1:90,1] + -0.762;
   1:  PR[GP1:91,2] = PR[GP1:90,2] + -23.500;
   1:L PR[91] R[100]mm/sec CNT100;
   1:  PR[GP1:91,1] = PR[GP1:90,1] + -0.352;
   1:  PR[GP1:91,2] = PR[GP1:90,2] + -23.464;
   1:L PR[91] R[100]mm/sec CNT100;
   1:  PR[GP1:91,1] = PR[GP1:90,1] + 0.519;
   1:L PR[91] R[100]mm/sec CNT100;
   1:  PR[GP1:91,1] = PR[GP1:90,1] + 7.079;
   1:  PR[GP1:91,2] = PR[GP1:90,2] + -24.109;
   1:L PR[91] R[100]mm/sec CNT100;
   1:  PR[GP1:91,1] = PR[GP1:90,1] + 7.266;
   1:  PR[GP1:91,2] = PR[GP1:90,2] + -24.085;
   1:L PR[91] R[100]mm/sec CNT100;
   1:  PR[GP1:91,1] = PR[GP1:90,1] + 13.297;
   1:  PR[GP1:91,2] = PR[GP1:90,2] + -23.125;
   1:L PR[91] R[100]mm/sec CNT100;
   1:  PR[GP1:91,1] = PR[GP1:90,1] + 13.701;
   1:  PR[GP1:91,2] = PR[GP1:90,2] + -22.963;
   1:L PR[91] R[100]mm/sec CNT100;
   1:  PR[GP1:91,1] = PR[GP1:90,1] + 19.048;
   1:  PR[GP1:91,2] = PR[GP1:90,2] + -20.638;
   1:L PR[91] R[100]mm/sec CNT100;
   1:  PR[GP1:91,1] = PR[GP1:90,1] + 19.581;
   1:  PR[GP1:91,2] = PR[GP1:90,2] + -20.242;
   1:L PR[91] R[100]mm/sec CNT100;
   1:  PR[GP1:91,1] = PR[GP1:90,1] + 23.948;
   1:  PR[GP1:91,2] = PR[GP1:90,2] + -16.826;
   1:L PR[91] R[100]mm/sec CNT100;
   1:  PR[GP1:91,1] = PR[GP1:90,1] + 24.480;
   1:  PR[GP1:91,2] = PR[GP1:90,2] + -16.155;
   1:L PR[91] R[100]mm/sec CNT100;
   1:  PR[GP1:91,1] = PR[GP1:90,1] + 27.690;
   1:  PR[GP1:91,2] = PR[GP1:90,2] + -11.931;
   1:L PR[91] R[100]mm/sec CNT100;
   1:  PR[GP1:91,1] = PR[GP1:90,1] + 28.081;
   1:  PR[GP1:91,2] = PR[GP1:90,2] + -11.033;
   1:L PR[91] R[100]mm/sec CNT100;
   1:  PR[GP1:91,1] = PR[GP1:90,1] + 30.029;
   1:  PR[GP1:91,2] = PR[GP1:90,2] + -6.338;
   1:L PR[91] R[100]mm/sec CNT100;
   1:  PR[GP1:91,1] = PR[GP1:90,1] + 30.171;
   1:  PR[GP1:91,2] = PR[GP1:90,2] + -5.288;
   1:L PR[91] R[100]mm/sec CNT100;
   1:  PR[GP1:91,1] = PR[GP1:90,1] + 30.322;
   1:  PR[GP1:91,2] = PR[GP1:90,2] + -3.763;
   1:L PR[91] R[100]mm/sec CNT100;
   1:  PR[GP1:91,1] = PR[GP1:90,1] + 30.779;
   1:  PR[GP1:91,2] = PR[GP1:90,2] + -0.286;
   1:L PR[91] R[100]mm/sec CNT100;
   1:  PR[GP1:91,1] = PR[GP1:90,1] + 30.675;
   1:  PR[GP1:91,2] = PR[GP1:90,2] + 0.805;
   1:L PR[91] R[100]mm/sec CNT100;
   1:  PR[GP1:91,1] = PR[GP1:90,1] + 30.029;
   1:  PR[GP1:91,2] = PR[GP1:90,2] + 5.711;
   1:L PR[91] R[100]mm/sec CNT100;
   1:  PR[GP1:91,1] = PR[GP1:90,1] + 28.086;
   1:  PR[GP1:91,2] = PR[GP1:90,2] + 10.399;
   1:L PR[91] R[100]mm/sec CNT100;
   1:  PR[GP1:91,1] = PR[GP1:90,1] + 27.696;
   1:  PR[GP1:91,2] = PR[GP1:90,2] + 11.297;
   1:L PR[91] R[100]mm/sec CNT100;
   1:  PR[GP1:91,1] = PR[GP1:90,1] + 24.491;
   1:  PR[GP1:91,2] = PR[GP1:90,2] + 15.518;
   1:L PR[91] R[100]mm/sec CNT100;
   1:  PR[GP1:91,1] = PR[GP1:90,1] + 23.961;
   1:  PR[GP1:91,2] = PR[GP1:90,2] + 16.189;
   1:L PR[91] R[100]mm/sec CNT100;
   1:  PR[GP1:91,1] = PR[GP1:90,1] + 19.601;
   1:  PR[GP1:91,2] = PR[GP1:90,2] + 19.606;
   1:L PR[91] R[100]mm/sec CNT100;
   1:  PR[GP1:91,1] = PR[GP1:90,1] + 19.069;
   1:  PR[GP1:91,2] = PR[GP1:90,2] + 20.001;
   1:L PR[91] R[100]mm/sec CNT100;
   1:  PR[GP1:91,1] = PR[GP1:90,1] + 13.731;
   1:  PR[GP1:91,2] = PR[GP1:90,2] + 22.330;
   1:L PR[91] R[100]mm/sec CNT100;
   1:  PR[GP1:91,1] = PR[GP1:90,1] + 13.326;
   1:  PR[GP1:91,2] = PR[GP1:90,2] + 22.493;
   1:L PR[91] R[100]mm/sec CNT100;
   1:  PR[GP1:91,1] = PR[GP1:90,1] + 7.303;
   1:  PR[GP1:91,2] = PR[GP1:90,2] + 23.459;
   1:L PR[91] R[100]mm/sec CNT100;
   1:  PR[GP1:91,1] = PR[GP1:90,1] + 7.115;
   1:  PR[GP1:91,2] = PR[GP1:90,2] + 23.484;
   1:L PR[91] R[100]mm/sec CNT100;
   1:  PR[GP1:91,1] = PR[GP1:90,1] + 0.518;
   1:  PR[GP1:91,2] = PR[GP1:90,2] + 22.840;
   1:L PR[91] R[100]mm/sec CNT100;
   1:  PR[91] = PR[90];
   1:  PR[GP1:91,1] = PR[GP1:90,1] + -0.337;
   1:  PR[GP1:91,2] = PR[GP1:90,2] + 23.004;
   1:  PR[GP1:91,3] = PR[GP1:90,3] + 58.255;
   1:L PR[91] R[100]mm/sec CNT100;
   1:  PR[GP1:91,1] = PR[GP1:90,1] + -4.502;
   1:  PR[GP1:91,2] = PR[GP1:90,2] + 23.366;
   1:L PR[91] R[100]mm/sec CNT100;
   1:  PR[GP1:91,1] = PR[GP1:90,1] + -6.737;
   1:  PR[GP1:91,2] = PR[GP1:90,2] + 23.581;
   1:L PR[91] R[100]mm/sec CNT100;
   1:  PR[GP1:91,1] = PR[GP1:90,1] + -12.984;
   1:  PR[GP1:91,2] = PR[GP1:90,2] + 22.584;
   1:L PR[91] R[100]mm/sec CNT100;
   1:  PR[GP1:91,1] = PR[GP1:90,1] + -13.148;
   1:  PR[GP1:91,2] = PR[GP1:90,2] + 22.517;
   1:L PR[91] R[100]mm/sec CNT100;
   1:  PR[GP1:91,1] = PR[GP1:90,1] + -18.739;
   1:  PR[GP1:91,2] = PR[GP1:90,2] + 20.078;
   1:L PR[91] R[100]mm/sec CNT100;
   1:  PR[GP1:91,1] = PR[GP1:90,1] + -19.061;
   1:  PR[GP1:91,2] = PR[GP1:90,2] + 19.839;
   1:L PR[91] R[100]mm/sec CNT100;
   1:  PR[GP1:91,1] = PR[GP1:90,1] + -23.642;
   1:  PR[GP1:91,2] = PR[GP1:90,2] + 16.250;
   1:L PR[91] R[100]mm/sec CNT100;
   1:  PR[GP1:91,1] = PR[GP1:90,1] + -24.009;
   1:  PR[GP1:91,2] = PR[GP1:90,2] + 15.787;
   1:L PR[91] R[100]mm/sec CNT100;
   1:  PR[GP1:91,1] = PR[GP1:90,1] + -27.384;
   1:  PR[GP1:91,2] = PR[GP1:90,2] + 11.344;
   1:L PR[91] R[100]mm/sec CNT100;
   1:  PR[GP1:91,1] = PR[GP1:90,1] + -27.671;
   1:  PR[GP1:91,2] = PR[GP1:90,2] + 10.681;
   1:L PR[91] R[100]mm/sec CNT100;
   1:  PR[GP1:91,1] = PR[GP1:90,1] + -29.723;
   1:  PR[GP1:91,2] = PR[GP1:90,2] + 5.722;
   1:L PR[91] R[100]mm/sec CNT100;
   1:  PR[GP1:91,1] = PR[GP1:90,1] + -29.830;
   1:  PR[GP1:91,2] = PR[GP1:90,2] + 4.936;
   1:L PR[91] R[100]mm/sec CNT100;
   1:  PR[GP1:91,1] = PR[GP1:90,1] + -29.949;
   1:  PR[GP1:91,2] = PR[GP1:90,2] + 3.729;
   1:L PR[91] R[100]mm/sec CNT100;
   1:  PR[GP1:91,1] = PR[GP1:90,1] + -30.483;
   1:  PR[GP1:91,2] = PR[GP1:90,2] + -0.338;
   1:L PR[91] R[100]mm/sec CNT100;
   1:  PR[GP1:91,1] = PR[GP1:90,1] + -30.403;
   1:  PR[GP1:91,2] = PR[GP1:90,2] + -1.175;
   1:L PR[91] R[100]mm/sec CNT100;
   1:  PR[GP1:91,1] = PR[GP1:90,1] + -29.720;
   1:  PR[GP1:91,2] = PR[GP1:90,2] + -6.354;
   1:L PR[91] R[100]mm/sec CNT100;
   1:  PR[GP1:91,1] = PR[GP1:90,1] + -27.665;
   1:  PR[GP1:91,2] = PR[GP1:90,2] + -11.315;
   1:L PR[91] R[100]mm/sec CNT100;
   1:  PR[GP1:91,1] = PR[GP1:90,1] + -27.378;
   1:  PR[GP1:91,2] = PR[GP1:90,2] + -11.978;
   1:L PR[91] R[100]mm/sec CNT100;
   1:  PR[GP1:91,1] = PR[GP1:90,1] + -23.997;
   1:  PR[GP1:91,2] = PR[GP1:90,2] + -16.424;
   1:L PR[91] R[100]mm/sec CNT100;
   1:  PR[GP1:91,1] = PR[GP1:90,1] + -23.630;
   1:  PR[GP1:91,2] = PR[GP1:90,2] + -16.886;
   1:L PR[91] R[100]mm/sec CNT100;
   1:  PR[GP1:91,1] = PR[GP1:90,1] + -19.040;
   1:  PR[GP1:91,2] = PR[GP1:90,2] + -20.476;
   1:L PR[91] R[100]mm/sec CNT100;
   1:  PR[GP1:91,1] = PR[GP1:90,1] + -18.719;
   1:  PR[GP1:91,2] = PR[GP1:90,2] + -20.714;
   1:L PR[91] R[100]mm/sec CNT100;
   1:  PR[GP1:91,1] = PR[GP1:90,1] + -12.936;
   1:  PR[GP1:91,2] = PR[GP1:90,2] + -23.219;
   1:L PR[91] R[100]mm/sec CNT100;
   1:  PR[GP1:91,1] = PR[GP1:90,1] + -6.715;
   1:  PR[GP1:91,2] = PR[GP1:90,2] + -24.208;
   1:L PR[91] R[100]mm/sec CNT100;
   1:  PR[GP1:91,1] = PR[GP1:90,1] + -4.834;
   1:  PR[GP1:91,2] = PR[GP1:90,2] + -24.022;
   1:L PR[91] R[100]mm/sec CNT100;
   1:  PR[GP1:91,1] = PR[GP1:90,1] + -0.338;
   1:  PR[GP1:91,2] = PR[GP1:90,2] + -23.626;
   1:L PR[91] R[100]mm/sec CNT100;
   1:  PR[GP1:91,1] = PR[GP1:90,1] + 0.497;
   1:L PR[91] R[100]mm/sec CNT100;
   1:  PR[GP1:91,1] = PR[GP1:90,1] + 4.986;
   1:  PR[GP1:91,2] = PR[GP1:90,2] + -24.021;
   1:L PR[91] R[100]mm/sec CNT100;
   1:  PR[GP1:91,1] = PR[GP1:90,1] + 6.860;
   1:  PR[GP1:91,2] = PR[GP1:90,2] + -24.206;
   1:L PR[91] R[100]mm/sec CNT100;
   1:  PR[GP1:91,1] = PR[GP1:90,1] + 13.114;
   1:  PR[GP1:91,2] = PR[GP1:90,2] + -23.215;
   1:L PR[91] R[100]mm/sec CNT100;
   1:  PR[GP1:91,1] = PR[GP1:90,1] + 13.277;
   1:  PR[GP1:91,2] = PR[GP1:90,2] + -23.149;
   1:L PR[91] R[100]mm/sec CNT100;
   1:  PR[GP1:91,1] = PR[GP1:90,1] + 18.876;
   1:  PR[GP1:91,2] = PR[GP1:90,2] + -20.714;
   1:L PR[91] R[100]mm/sec CNT100;
   1:  PR[GP1:91,1] = PR[GP1:90,1] + 19.198;
   1:  PR[GP1:91,2] = PR[GP1:90,2] + -20.476;
   1:L PR[91] R[100]mm/sec CNT100;
   1:  PR[GP1:91,1] = PR[GP1:90,1] + 23.786;
   1:  PR[GP1:91,2] = PR[GP1:90,2] + -16.886;
   1:L PR[91] R[100]mm/sec CNT100;
   1:  PR[GP1:91,1] = PR[GP1:90,1] + 24.154;
   1:  PR[GP1:91,2] = PR[GP1:90,2] + -16.423;
   1:L PR[91] R[100]mm/sec CNT100;
   1:  PR[GP1:91,1] = PR[GP1:90,1] + 27.535;
   1:  PR[GP1:91,2] = PR[GP1:90,2] + -11.974;
   1:L PR[91] R[100]mm/sec CNT100;
   1:  PR[GP1:91,1] = PR[GP1:90,1] + 27.823;
   1:  PR[GP1:91,2] = PR[GP1:90,2] + -11.313;
   1:L PR[91] R[100]mm/sec CNT100;
   1:  PR[GP1:91,1] = PR[GP1:90,1] + 29.878;
   1:  PR[GP1:91,2] = PR[GP1:90,2] + -6.359;
   1:L PR[91] R[100]mm/sec CNT100;
   1:  PR[GP1:91,1] = PR[GP1:90,1] + 29.985;
   1:  PR[GP1:91,2] = PR[GP1:90,2] + -5.569;
   1:L PR[91] R[100]mm/sec CNT100;
   1:  PR[GP1:91,1] = PR[GP1:90,1] + 30.105;
   1:  PR[GP1:91,2] = PR[GP1:90,2] + -4.360;
   1:L PR[91] R[100]mm/sec CNT100;
   1:  PR[GP1:91,1] = PR[GP1:90,1] + 30.640;
   1:  PR[GP1:91,2] = PR[GP1:90,2] + -0.286;
   1:L PR[91] R[100]mm/sec CNT100;
   1:  PR[GP1:91,1] = PR[GP1:90,1] + 30.560;
   1:  PR[GP1:91,2] = PR[GP1:90,2] + 0.553;
   1:L PR[91] R[100]mm/sec CNT100;
   1:  PR[GP1:91,1] = PR[GP1:90,1] + 29.879;
   1:  PR[GP1:91,2] = PR[GP1:90,2] + 5.731;
   1:L PR[91] R[100]mm/sec CNT100;
   1:  PR[GP1:91,1] = PR[GP1:90,1] + 27.828;
   1:  PR[GP1:91,2] = PR[GP1:90,2] + 10.679;
   1:L PR[91] R[100]mm/sec CNT100;
   1:  PR[GP1:91,1] = PR[GP1:90,1] + 27.541;
   1:  PR[GP1:91,2] = PR[GP1:90,2] + 11.339;
   1:L PR[91] R[100]mm/sec CNT100;
   1:  PR[GP1:91,1] = PR[GP1:90,1] + 24.166;
   1:  PR[GP1:91,2] = PR[GP1:90,2] + 15.786;
   1:L PR[91] R[100]mm/sec CNT100;
   1:  PR[GP1:91,1] = PR[GP1:90,1] + 23.799;
   1:  PR[GP1:91,2] = PR[GP1:90,2] + 16.250;
   1:L PR[91] R[100]mm/sec CNT100;
   1:  PR[GP1:91,1] = PR[GP1:90,1] + 19.219;
   1:  PR[GP1:91,2] = PR[GP1:90,2] + 19.839;
   1:L PR[91] R[100]mm/sec CNT100;
   1:  PR[GP1:91,1] = PR[GP1:90,1] + 18.897;
   1:  PR[GP1:91,2] = PR[GP1:90,2] + 20.078;
   1:L PR[91] R[100]mm/sec CNT100;
   1:  PR[GP1:91,1] = PR[GP1:90,1] + 13.123;
   1:  PR[GP1:91,2] = PR[GP1:90,2] + 22.586;
   1:L PR[91] R[100]mm/sec CNT100;
   1:  PR[GP1:91,1] = PR[GP1:90,1] + 6.909;
   1:  PR[GP1:91,2] = PR[GP1:90,2] + 23.583;
   1:L PR[91] R[100]mm/sec CNT100;
   1:  PR[GP1:91,1] = PR[GP1:90,1] + 4.657;
   1:  PR[GP1:91,2] = PR[GP1:90,2] + 23.365;
   1:L PR[91] R[100]mm/sec CNT100;
   1:  PR[GP1:91,1] = PR[GP1:90,1] + 0.496;
   1:  PR[GP1:91,2] = PR[GP1:90,2] + 23.004;
   1:L PR[91] R[100]mm/sec CNT100;
   1:  PR[91] = PR[90];
   1:  PR[GP1:91,1] = PR[GP1:90,1] + -0.323;
   1:  PR[GP1:91,2] = PR[GP1:90,2] + 23.167;
   1:  PR[GP1:91,3] = PR[GP1:90,3] + 58.865;
   1:L PR[91] R[100]mm/sec CNT100;
   1:  PR[GP1:91,1] = PR[GP1:90,1] + -6.498;
   1:  PR[GP1:91,2] = PR[GP1:90,2] + 23.701;
   1:L PR[91] R[100]mm/sec CNT100;
   1:  PR[GP1:91,1] = PR[GP1:90,1] + -12.789;
   1:  PR[GP1:91,2] = PR[GP1:90,2] + 22.676;
   1:L PR[91] R[100]mm/sec CNT100;
   1:  PR[GP1:91,1] = PR[GP1:90,1] + -18.550;
   1:  PR[GP1:91,2] = PR[GP1:90,2] + 20.162;
   1:L PR[91] R[100]mm/sec CNT100;
   1:  PR[GP1:91,1] = PR[GP1:90,1] + -23.470;
   1:  PR[GP1:91,2] = PR[GP1:90,2] + 16.318;
   1:L PR[91] R[100]mm/sec CNT100;
   1:  PR[GP1:91,1] = PR[GP1:90,1] + -27.223;
   1:  PR[GP1:91,2] = PR[GP1:90,2] + 11.393;
   1:L PR[91] R[100]mm/sec CNT100;
   1:  PR[GP1:91,1] = PR[GP1:90,1] + -29.573;
   1:  PR[GP1:91,2] = PR[GP1:90,2] + 5.742;
   1:L PR[91] R[100]mm/sec CNT100;
   1:  PR[GP1:91,1] = PR[GP1:90,1] + -29.644;
   1:  PR[GP1:91,2] = PR[GP1:90,2] + 5.217;
   1:L PR[91] R[100]mm/sec CNT100;
   1:  PR[GP1:91,1] = PR[GP1:90,1] + -29.732;
   1:  PR[GP1:91,2] = PR[GP1:90,2] + 4.326;
   1:L PR[91] R[100]mm/sec CNT100;
   1:  PR[GP1:91,1] = PR[GP1:90,1] + -30.345;
   1:  PR[GP1:91,2] = PR[GP1:90,2] + -0.338;
   1:L PR[91] R[100]mm/sec CNT100;
   1:  PR[GP1:91,1] = PR[GP1:90,1] + -30.289;
   1:  PR[GP1:91,2] = PR[GP1:90,2] + -0.923;
   1:L PR[91] R[100]mm/sec CNT100;
   1:  PR[GP1:91,1] = PR[GP1:90,1] + -29.570;
   1:  PR[GP1:91,2] = PR[GP1:90,2] + -6.374;
   1:L PR[91] R[100]mm/sec CNT100;
   1:  PR[GP1:91,1] = PR[GP1:90,1] + -27.217;
   1:  PR[GP1:91,2] = PR[GP1:90,2] + -12.029;
   1:L PR[91] R[100]mm/sec CNT100;
   1:  PR[GP1:91,1] = PR[GP1:90,1] + -23.670;
   1:  PR[GP1:91,2] = PR[GP1:90,2] + -16.691;
   1:L PR[91] R[100]mm/sec CNT100;
   1:  PR[GP1:91,1] = PR[GP1:90,1] + -23.468;
   1:  PR[GP1:91,2] = PR[GP1:90,2] + -16.946;
   1:L PR[91] R[100]mm/sec CNT100;
   1:  PR[GP1:91,1] = PR[GP1:90,1] + -18.530;
   1:  PR[GP1:91,2] = PR[GP1:90,2] + -20.798;
   1:L PR[91] R[100]mm/sec CNT100;
   1:  PR[GP1:91,1] = PR[GP1:90,1] + -12.751;
   1:  PR[GP1:91,2] = PR[GP1:90,2] + -23.309;
   1:L PR[91] R[100]mm/sec CNT100;
   1:  PR[GP1:91,1] = PR[GP1:90,1] + -10.118;
   1:  PR[GP1:91,2] = PR[GP1:90,2] + -23.728;
   1:L PR[91] R[100]mm/sec CNT100;
   1:  PR[GP1:91,1] = PR[GP1:90,1] + -6.477;
   1:  PR[GP1:91,2] = PR[GP1:90,2] + -24.330;
   1:L PR[91] R[100]mm/sec CNT100;
   1:  PR[GP1:91,1] = PR[GP1:90,1] + -6.453;
   1:  PR[GP1:91,2] = PR[GP1:90,2] + -24.328;
   1:L PR[91] R[100]mm/sec CNT100;
   1:  PR[GP1:91,1] = PR[GP1:90,1] + -0.324;
   1:  PR[GP1:91,2] = PR[GP1:90,2] + -23.789;
   1:L PR[91] R[100]mm/sec CNT100;
   1:  PR[GP1:91,1] = PR[GP1:90,1] + 0.483;
   1:L PR[91] R[100]mm/sec CNT100;
   1:  PR[GP1:91,1] = PR[GP1:90,1] + 6.583;
   1:  PR[GP1:91,2] = PR[GP1:90,2] + -24.325;
   1:L PR[91] R[100]mm/sec CNT100;
   1:  PR[GP1:91,1] = PR[GP1:90,1] + 6.654;
   1:  PR[GP1:91,2] = PR[GP1:90,2] + -24.328;
   1:L PR[91] R[100]mm/sec CNT100;
   1:  PR[GP1:91,1] = PR[GP1:90,1] + 10.266;
   1:  PR[GP1:91,2] = PR[GP1:90,2] + -23.729;
   1:L PR[91] R[100]mm/sec CNT100;
   1:  PR[GP1:91,1] = PR[GP1:90,1] + 12.910;
   1:  PR[GP1:91,2] = PR[GP1:90,2] + -23.308;
   1:L PR[91] R[100]mm/sec CNT100;
   1:  PR[GP1:91,1] = PR[GP1:90,1] + 18.688;
   1:  PR[GP1:91,2] = PR[GP1:90,2] + -20.798;
   1:L PR[91] R[100]mm/sec CNT100;
   1:  PR[GP1:91,1] = PR[GP1:90,1] + 23.615;
   1:  PR[GP1:91,2] = PR[GP1:90,2] + -16.954;
   1:L PR[91] R[100]mm/sec CNT100;
   1:  PR[GP1:91,1] = PR[GP1:90,1] + 27.374;
   1:  PR[GP1:91,2] = PR[GP1:90,2] + -12.024;
   1:L PR[91] R[100]mm/sec CNT100;
   1:  PR[GP1:91,1] = PR[GP1:90,1] + 29.728;
   1:  PR[GP1:91,2] = PR[GP1:90,2] + -6.378;
   1:L PR[91] R[100]mm/sec CNT100;
   1:  PR[GP1:91,1] = PR[GP1:90,1] + 29.799;
   1:  PR[GP1:91,2] = PR[GP1:90,2] + -5.851;
   1:L PR[91] R[100]mm/sec CNT100;
   1:  PR[GP1:91,1] = PR[GP1:90,1] + 29.888;
   1:  PR[GP1:91,2] = PR[GP1:90,2] + -4.958;
   1:L PR[91] R[100]mm/sec CNT100;
   1:  PR[GP1:91,1] = PR[GP1:90,1] + 30.502;
   1:  PR[GP1:91,2] = PR[GP1:90,2] + -0.286;
   1:L PR[91] R[100]mm/sec CNT100;
   1:  PR[GP1:91,1] = PR[GP1:90,1] + 30.446;
   1:  PR[GP1:91,2] = PR[GP1:90,2] + 0.301;
   1:L PR[91] R[100]mm/sec CNT100;
   1:  PR[GP1:91,1] = PR[GP1:90,1] + 29.728;
   1:  PR[GP1:91,2] = PR[GP1:90,2] + 5.751;
   1:L PR[91] R[100]mm/sec CNT100;
   1:  PR[GP1:91,1] = PR[GP1:90,1] + 27.380;
   1:  PR[GP1:91,2] = PR[GP1:90,2] + 11.390;
   1:L PR[91] R[100]mm/sec CNT100;
   1:  PR[GP1:91,1] = PR[GP1:90,1] + 23.627;
   1:  PR[GP1:91,2] = PR[GP1:90,2] + 16.318;
   1:L PR[91] R[100]mm/sec CNT100;
   1:  PR[GP1:91,1] = PR[GP1:90,1] + 18.708;
   1:  PR[GP1:91,2] = PR[GP1:90,2] + 20.162;
   1:L PR[91] R[100]mm/sec CNT100;
   1:  PR[GP1:91,1] = PR[GP1:90,1] + 12.938;
   1:  PR[GP1:91,2] = PR[GP1:90,2] + 22.676;
   1:L PR[91] R[100]mm/sec CNT100;
   1:  PR[GP1:91,1] = PR[GP1:90,1] + 10.264;
   1:  PR[GP1:91,2] = PR[GP1:90,2] + 23.105;
   1:L PR[91] R[100]mm/sec CNT100;
   1:  PR[GP1:91,1] = PR[GP1:90,1] + 6.673;
   1:  PR[GP1:91,2] = PR[GP1:90,2] + 23.704;
   1:L PR[91] R[100]mm/sec CNT100;
   1:  PR[GP1:91,1] = PR[GP1:90,1] + 6.540;
   1:  PR[GP1:91,2] = PR[GP1:90,2] + 23.694;
   1:L PR[91] R[100]mm/sec CNT100;
   1:  PR[GP1:91,1] = PR[GP1:90,1] + 0.482;
   1:  PR[GP1:91,2] = PR[GP1:90,2] + 23.167;
   1:L PR[91] R[100]mm/sec CNT100;
   1:  PR[91] = PR[90];
   1:  PR[GP1:91,1] = PR[GP1:90,1] + -0.308;
   1:  PR[GP1:91,2] = PR[GP1:90,2] + 23.330;
   1:  PR[GP1:91,3] = PR[GP1:90,3] + 59.475;
   1:L PR[91] R[100]mm/sec CNT100;
   1:  PR[GP1:91,1] = PR[GP1:90,1] + -6.267;
   1:  PR[GP1:91,2] = PR[GP1:90,2] + 23.841;
   1:L PR[91] R[100]mm/sec CNT100;
   1:  PR[GP1:91,1] = PR[GP1:90,1] + -6.497;
   1:  PR[GP1:91,2] = PR[GP1:90,2] + 23.813;
   1:L PR[91] R[100]mm/sec CNT100;
   1:  PR[GP1:91,1] = PR[GP1:90,1] + -12.584;
   1:  PR[GP1:91,2] = PR[GP1:90,2] + 22.798;
   1:L PR[91] R[100]mm/sec CNT100;
   1:  PR[GP1:91,1] = PR[GP1:90,1] + -18.375;
   1:  PR[GP1:91,2] = PR[GP1:90,2] + 20.241;
   1:L PR[91] R[100]mm/sec CNT100;
   1:  PR[GP1:91,1] = PR[GP1:90,1] + -23.307;
   1:  PR[GP1:91,2] = PR[GP1:90,2] + 16.380;
   1:L PR[91] R[100]mm/sec CNT100;
   1:  PR[GP1:91,1] = PR[GP1:90,1] + -27.068;
   1:  PR[GP1:91,2] = PR[GP1:90,2] + 11.437;
   1:L PR[91] R[100]mm/sec CNT100;
   1:  PR[GP1:91,1] = PR[GP1:90,1] + -29.417;
   1:  PR[GP1:91,2] = PR[GP1:90,2] + 5.777;
   1:L PR[91] R[100]mm/sec CNT100;
   1:  PR[GP1:91,1] = PR[GP1:90,1] + -29.517;
   1:  PR[GP1:91,2] = PR[GP1:90,2] + 4.910;
   1:L PR[91] R[100]mm/sec CNT100;
   1:  PR[GP1:91,1] = PR[GP1:90,1] + -30.206;
   1:  PR[GP1:91,2] = PR[GP1:90,2] + -0.338;
   1:L PR[91] R[100]mm/sec CNT100;
   1:  PR[GP1:91,1] = PR[GP1:90,1] + -30.174;
   1:  PR[GP1:91,2] = PR[GP1:90,2] + -0.671;
   1:L PR[91] R[100]mm/sec CNT100;
   1:  PR[GP1:91,1] = PR[GP1:90,1] + -29.420;
   1:  PR[GP1:91,2] = PR[GP1:90,2] + -6.396;
   1:L PR[91] R[100]mm/sec CNT100;
   1:  PR[GP1:91,1] = PR[GP1:90,1] + -27.062;
   1:  PR[GP1:91,2] = PR[GP1:90,2] + -12.071;
   1:L PR[91] R[100]mm/sec CNT100;
   1:  PR[GP1:91,1] = PR[GP1:90,1] + -23.345;
   1:  PR[GP1:91,2] = PR[GP1:90,2] + -16.958;
   1:L PR[91] R[100]mm/sec CNT100;
   1:  PR[GP1:91,1] = PR[GP1:90,1] + -23.305;
   1:  PR[GP1:91,2] = PR[GP1:90,2] + -17.008;
   1:L PR[91] R[100]mm/sec CNT100;
   1:  PR[GP1:91,1] = PR[GP1:90,1] + -18.355;
   1:  PR[GP1:91,2] = PR[GP1:90,2] + -20.877;
   1:L PR[91] R[100]mm/sec CNT100;
   1:  PR[GP1:91,1] = PR[GP1:90,1] + -12.520;
   1:  PR[GP1:91,2] = PR[GP1:90,2] + -23.437;
   1:L PR[91] R[100]mm/sec CNT100;
   1:  PR[GP1:91,1] = PR[GP1:90,1] + -6.461;
   1:  PR[GP1:91,2] = PR[GP1:90,2] + -24.439;
   1:L PR[91] R[100]mm/sec CNT100;
   1:  PR[GP1:91,1] = PR[GP1:90,1] + -6.228;
   1:  PR[GP1:91,2] = PR[GP1:90,2] + -24.466;
   1:L PR[91] R[100]mm/sec CNT100;
   1:  PR[GP1:91,1] = PR[GP1:90,1] + -0.309;
   1:  PR[GP1:91,2] = PR[GP1:90,2] + -23.951;
   1:L PR[91] R[100]mm/sec CNT100;
   1:  PR[GP1:91,1] = PR[GP1:90,1] + 0.468;
   1:L PR[91] R[100]mm/sec CNT100;
   1:  PR[GP1:91,1] = PR[GP1:90,1] + 6.009;
   1:  PR[GP1:91,2] = PR[GP1:90,2] + -24.438;
   1:L PR[91] R[100]mm/sec CNT100;
   1:  PR[GP1:91,1] = PR[GP1:90,1] + 6.422;
   1:  PR[GP1:91,2] = PR[GP1:90,2] + -24.471;
   1:L PR[91] R[100]mm/sec CNT100;
   1:  PR[GP1:91,1] = PR[GP1:90,1] + 6.467;
   1:  PR[GP1:91,2] = PR[GP1:90,2] + -24.468;
   1:L PR[91] R[100]mm/sec CNT100;
   1:  PR[GP1:91,1] = PR[GP1:90,1] + 12.685;
   1:  PR[GP1:91,2] = PR[GP1:90,2] + -23.435;
   1:L PR[91] R[100]mm/sec CNT100;
   1:  PR[GP1:91,1] = PR[GP1:90,1] + 18.513;
   1:  PR[GP1:91,2] = PR[GP1:90,2] + -20.877;
   1:L PR[91] R[100]mm/sec CNT100;
   1:  PR[GP1:91,1] = PR[GP1:90,1] + 23.452;
   1:  PR[GP1:91,2] = PR[GP1:90,2] + -17.016;
   1:L PR[91] R[100]mm/sec CNT100;
   1:  PR[GP1:91,1] = PR[GP1:90,1] + 27.219;
   1:  PR[GP1:91,2] = PR[GP1:90,2] + -12.068;
   1:L PR[91] R[100]mm/sec CNT100;
   1:  PR[GP1:91,1] = PR[GP1:90,1] + 29.572;
   1:  PR[GP1:91,2] = PR[GP1:90,2] + -6.412;
   1:L PR[91] R[100]mm/sec CNT100;
   1:  PR[GP1:91,1] = PR[GP1:90,1] + 29.672;
   1:  PR[GP1:91,2] = PR[GP1:90,2] + -5.544;
   1:L PR[91] R[100]mm/sec CNT100;
   1:  PR[GP1:91,1] = PR[GP1:90,1] + 30.363;
   1:  PR[GP1:91,2] = PR[GP1:90,2] + -0.286;
   1:L PR[91] R[100]mm/sec CNT100;
   1:  PR[GP1:91,1] = PR[GP1:90,1] + 30.331;
   1:  PR[GP1:91,2] = PR[GP1:90,2] + 0.048;
   1:L PR[91] R[100]mm/sec CNT100;
   1:  PR[GP1:91,1] = PR[GP1:90,1] + 29.578;
   1:  PR[GP1:91,2] = PR[GP1:90,2] + 5.772;
   1:L PR[91] R[100]mm/sec CNT100;
   1:  PR[GP1:91,1] = PR[GP1:90,1] + 27.225;
   1:  PR[GP1:91,2] = PR[GP1:90,2] + 11.433;
   1:L PR[91] R[100]mm/sec CNT100;
   1:  PR[GP1:91,1] = PR[GP1:90,1] + 23.464;
   1:  PR[GP1:91,2] = PR[GP1:90,2] + 16.379;
   1:L PR[91] R[100]mm/sec CNT100;
   1:  PR[GP1:91,1] = PR[GP1:90,1] + 18.533;
   1:  PR[GP1:91,2] = PR[GP1:90,2] + 20.241;
   1:L PR[91] R[100]mm/sec CNT100;
   1:  PR[GP1:91,1] = PR[GP1:90,1] + 12.712;
   1:  PR[GP1:91,2] = PR[GP1:90,2] + 22.803;
   1:L PR[91] R[100]mm/sec CNT100;
   1:  PR[GP1:91,1] = PR[GP1:90,1] + 6.655;
   1:  PR[GP1:91,2] = PR[GP1:90,2] + 23.813;
   1:L PR[91] R[100]mm/sec CNT100;
   1:  PR[GP1:91,1] = PR[GP1:90,1] + 6.426;
   1:  PR[GP1:91,2] = PR[GP1:90,2] + 23.842;
   1:L PR[91] R[100]mm/sec CNT100;
   1:  PR[GP1:91,1] = PR[GP1:90,1] + 0.466;
   1:  PR[GP1:91,2] = PR[GP1:90,2] + 23.331;
   1:L PR[91] R[100]mm/sec CNT100 TB   .50sec,CALL END_PUD;
   1:  DO[117:Laser Start]=OFF;
   1:  PR[92] = PR[91];
   1:  PR[GP1:92,3] = PR[GP1:92,3] + 50;
   1:J PR[92] 10% FINE;
   1:  WAIT   5.00(sec);
   1:  DO[119:Gas]=OFF;
   1:  CALL HOME_ALL;
/POS
/END
